KUKA KRL program: EPS_2_25369_MH4A_A_20251128065500.src

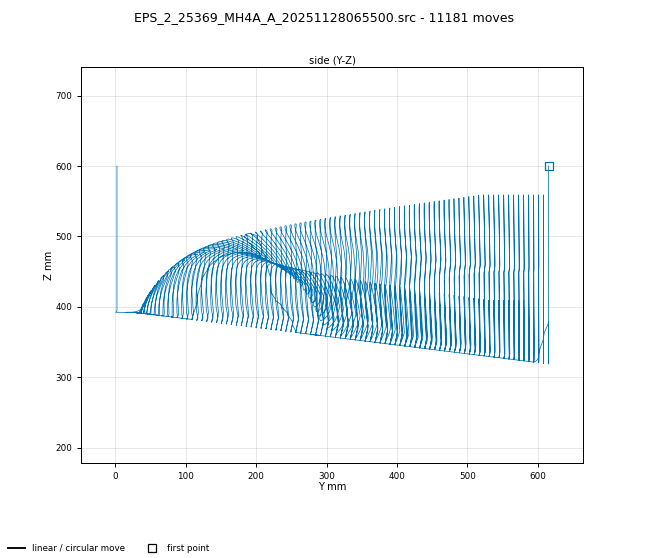
[picture p0: tool path of EPS_2_25369_MH4A_A_20251128065500.src, 11181 of 11183 moves have a stored position in this frame; points joined in program order, loops and branches not executed]
&ACCESS RVP
&REL 4
&COMMENT QRS 19112012
&PARAM EDITMASK = *
DEF PART()
EXT BAS (BAS_COMMAND :IN,REAL :IN )
INT I
BAS (#INITMOV,0 )

;KUKA QRS Post kuka4.cps  Date:22-06-2017 !

File_ID=2934

QRS_PRE_INIT()

;Init var - Until changes are made in qrs_pre_init
Outlet_Square_prg=0
Inlet_1_Square_prg=0
Inlet_2_Square_prg=0
Inlet_3_Square_prg=0
Inlet_4_Square_prg=0
Inlet_5_Square_prg=0

Outlet_1={X 0.000, Y 520.860, Z 458.500, B 0.000, E1 0.000 }
Inlet_1={X 0.000, Y 531.730, Z 308.500, B 0.000, E1 89.000 }
Outlet_1_type=201
Inlet_1_type=201
;QRS#1=Sidecore dimensions
;QRS#2=200-8" PVC SDR 35
;QRS#3=200-8" PVC SDR 35
;QRS#4=
;QRS#5=
;QRS#6=
;QRS#7=
;QRS#8=
;QRS#9=12-08 PSX
;QRS#10=12-08 PSX
;QRS#11=
;QRS#12=
;QRS#13=
;QRS#14=
;QRS#15=
;QRS#16=1220x127x838 2,75'
;QRS#17=EPS Height
;QRS#18=559
;QRS#19=*
;QRS#20= UPDATED VERSION 22-06-2017
;QRS#21=*
Outlet_Square=0100
Inlet_1_Square=0100
Inlet_2_Square=0
Inlet_3_Square=0
Inlet_4_Square=0
Inlet_5_Square=0
Mill_Square=1
Outlet_Square_Prg=204
Inlet_1_Square_prg=204

QRS_INIT()

$ADVANCE=5

; T1
PTP {E1 173.485,E2 173.485}
PTP {X 0,Y 615.499,A -85,B 0,C 180,E1 173.485,E2 173.485,E3 0,E4 0,E5 0,E6 0}
QRS_SPEED_INIT()
LIN {X 0,Y 615.499,Z 600,A -85,B 0,C 180,E1 173.485,E2 173.485,E3 0,E4 0,E5 0,E6 0} C_VEL
LIN {X 0,Y 615.499,Z 392.663,A -85,B 0,C 180,E1 173.485,E2 173.485} C_VEL
LIN {X 0,Y 615.499,Z 380.744,A -85,B 0,C 180,E1 173.485,E2 173.485} C_VEL
LIN {X 0,Y 615.497,Z 379.208,A -85,B 0,C 180,E1 173.418,E2 173.418} C_VEL
LIN {X 0,Y 615.498,Z 369.663,A -85,B 0,C 180,E1 172.455,E2 172.455} C_VEL
LIN {X 0,Y 615.497,Z 359.4,A -85,B 0,C 180,E1 171.629,E2 171.629} C_VEL
LIN {X 0,Y 615.486,Z 347.853,A -85,B 0,C 180,E1 170.884,E2 170.884} C_VEL
LIN {X 0,Y 615.482,Z 336.334,A -85,B 0,C 180,E1 170.304,E2 170.304} C_VEL
LIN {X 0,Y 615.493,Z 324.409,A -85,B 0,C 180,E1 169.847,E2 169.847} C_VEL
LIN {X 0,Y 615.489,Z 318.699,A -85,B 0,C 180,E1 169.66,E2 169.66} C_VEL
LIN {X 0,Y 615.494,Z 318.687,A -85,B 0,C 180,E1 166.799,E2 166.799} C_VEL
LIN {X 0,Y 615.488,Z 318.692,A -85,B 0,C 180,E1 164.095,E2 164.095} C_VEL
LIN {X 0,Y 615.477,Z 318.693,A -85,B 0,C 180,E1 161.354,E2 161.354} C_VEL
LIN {X 0,Y 615.479,Z 318.69,A -85,B 0,C 180,E1 158.568,E2 158.568} C_VEL
LIN {X 0,Y 615.496,Z 318.696,A -85,B 0,C 180,E1 155.728,E2 155.728} C_VEL
LIN {X 0,Y 615.491,Z 318.686,A -85,B 0,C 180,E1 152.823,E2 152.823} C_VEL
LIN {X 0,Y 615.488,Z 318.69,A -85,B 0,C 180,E1 149.84,E2 149.84} C_VEL
LIN {X 0,Y 615.477,Z 318.689,A -85,B 0,C 180,E1 147.542,E2 147.542} C_VEL
LIN {X 0,Y 615.49,Z 318.695,A -85,B 0,C 180,E1 145.185,E2 145.185} C_VEL
LIN {X 0,Y 615.479,Z 318.692,A -85,B 0,C 180,E1 142.757,E2 142.757} C_VEL
LIN {X 0,Y 615.493,Z 318.694,A -85,B 0,C 180,E1 139.911,E2 139.911} C_VEL
LIN {X 0,Y 615.483,Z 318.688,A -85,B 0,C 180,E1 136.954,E2 136.954} C_VEL
LIN {X 0,Y 615.482,Z 318.693,A -85,B 0,C 180,E1 133.997,E2 133.997} C_VEL
LIN {X 0,Y 615.488,Z 318.687,A -85,B 0,C 180,E1 131.474,E2 131.474} C_VEL
LIN {X 0,Y 615.489,Z 318.698,A -85,B 0,C 180,E1 128.905,E2 128.905} C_VEL
LIN {X 0,Y 615.485,Z 318.687,A -85,B 0,C 180,E1 126.425,E2 126.425} C_VEL
LIN {X 0,Y 615.498,Z 318.694,A -85,B 0,C 180,E1 123.536,E2 123.536} C_VEL
LIN {X 0,Y 615.478,Z 318.689,A -85,B 0,C 180,E1 120.92,E2 120.92} C_VEL
LIN {X 0,Y 615.498,Z 318.7,A -85,B 0,C 180,E1 118.452,E2 118.452} C_VEL
LIN {X 0,Y 615.498,Z 318.685,A -85,B 0,C 180,E1 115.571,E2 115.571} C_VEL
LIN {X 0,Y 615.493,Z 318.693,A -85,B 0,C 180,E1 112.844,E2 112.844} C_VEL
LIN {X 0,Y 615.479,Z 318.692,A -85,B 0,C 180,E1 110.033,E2 110.033} C_VEL
LIN {X 0,Y 615.477,Z 318.691,A -85,B 0,C 180,E1 107.271,E2 107.271} C_VEL
LIN {X 0,Y 615.494,Z 318.693,A -85,B 0,C 180,E1 104.549,E2 104.549} C_VEL
LIN {X 0,Y 615.489,Z 318.687,A -85,B 0,C 180,E1 101.861,E2 101.861} C_VEL
LIN {X 0,Y 615.483,Z 318.696,A -85,B 0,C 180,E1 99.199,E2 99.199} C_VEL
LIN {X 0,Y 615.479,Z 318.69,A -85,B 0,C 180,E1 96.557,E2 96.557} C_VEL
LIN {X 0,Y 615.491,Z 318.693,A -85,B 0,C 180,E1 93.928,E2 93.928} C_VEL
LIN {X 0,Y 615.48,Z 318.69,A -85,B 0,C 180,E1 91.309,E2 91.309} C_VEL
LIN {X 0,Y 615.489,Z 318.692,A -85,B 0,C 180,E1 88.691,E2 88.691} C_VEL
LIN {X 0,Y 615.49,Z 318.689,A -85,B 0,C 180,E1 86.071,E2 86.071} C_VEL
LIN {X 0,Y 615.48,Z 318.693,A -85,B 0,C 180,E1 83.428,E2 83.428} C_VEL
LIN {X 0,Y 615.479,Z 318.692,A -85,B 0,C 180,E1 80.801,E2 80.801} C_VEL
LIN {X 0,Y 615.491,Z 318.69,A -85,B 0,C 180,E1 78.139,E2 78.139} C_VEL
LIN {X 0,Y 615.485,Z 318.69,A -85,B 0,C 180,E1 75.451,E2 75.451} C_VEL
LIN {X 0,Y 615.479,Z 318.695,A -85,B 0,C 180,E1 72.729,E2 72.729} C_VEL
LIN {X 0,Y 615.479,Z 318.689,A -85,B 0,C 180,E1 69.967,E2 69.967} C_VEL
LIN {X 0,Y 615.494,Z 318.699,A -85,B 0,C 180,E1 67.155,E2 67.155} C_VEL
LIN {X 0,Y 615.488,Z 318.687,A -85,B 0,C 180,E1 64.284,E2 64.284} C_VEL
LIN {X 0,Y 615.486,Z 318.691,A -85,B 0,C 180,E1 61.342,E2 61.342} C_VEL
LIN {X 0,Y 615.479,Z 318.689,A -85,B 0,C 180,E1 58.915,E2 58.915} C_VEL
LIN {X 0,Y 615.498,Z 318.7,A -85,B 0,C 180,E1 56.464,E2 56.464} C_VEL
LIN {X 0,Y 615.488,Z 318.688,A -85,B 0,C 180,E1 53.575,E2 53.575} C_VEL
LIN {X 0,Y 615.494,Z 318.694,A -85,B 0,C 180,E1 50.937,E2 50.937} C_VEL
LIN {X 0,Y 615.487,Z 318.686,A -85,B 0,C 180,E1 48.526,E2 48.526} C_VEL
LIN {X 0,Y 615.497,Z 318.701,A -85,B 0,C 180,E1 45.851,E2 45.851} C_VEL
LIN {X 0,Y 615.483,Z 318.688,A -85,B 0,C 180,E1 43.046,E2 43.046} C_VEL
LIN {X 0,Y 615.493,Z 318.7,A -85,B 0,C 180,E1 40.606,E2 40.606} C_VEL
LIN {X 0,Y 615.483,Z 318.688,A -85,B 0,C 180,E1 38.011,E2 38.011} C_VEL
LIN {X 0,Y 615.487,Z 318.692,A -85,B 0,C 180,E1 35.616,E2 35.616} C_VEL
LIN {X 0,Y 615.492,Z 318.694,A -85,B 0,C 180,E1 33.236,E2 33.236} C_VEL
LIN {X 0,Y 615.488,Z 318.686,A -85,B 0,C 180,E1 30.92,E2 30.92} C_VEL
LIN {X 0,Y 615.485,Z 318.695,A -85,B 0,C 180,E1 28.449,E2 28.449} C_VEL
LIN {X 0,Y 615.478,Z 318.689,A -85,B 0,C 180,E1 25.716,E2 25.716} C_VEL
LIN {X 0,Y 615.473,Z 318.69,A -85,B 0,C 180,E1 23.557,E2 23.557} C_VEL
LIN {X 0,Y 615.48,Z 318.694,A -85,B 0,C 180,E1 21.432,E2 21.432} C_VEL
LIN {X 0,Y 615.476,Z 318.69,A -85,B 0,C 180,E1 18.646,E2 18.646} C_VEL
LIN {X 0,Y 615.491,Z 318.697,A -85,B 0,C 180,E1 15.905,E2 15.905} C_VEL
LIN {X 0,Y 615.494,Z 318.685,A -85,B 0,C 180,E1 13.201,E2 13.201} C_VEL
LIN {X 0,Y 615.495,Z 318.699,A -85,B 0,C 180,E1 10.527,E2 10.527} C_VEL
LIN {X 0,Y 615.478,Z 318.689,A -85,B 0,C 180,E1 7.876,E2 7.876} C_VEL
LIN {X 0,Y 615.495,Z 318.698,A -85,B 0,C 180,E1 5.241,E2 5.241} C_VEL
LIN {X 0,Y 615.488,Z 318.687,A -85,B 0,C 180,E1 2.618,E2 2.618} C_VEL
LIN {X 0,Y 615.493,Z 318.696,A -85,B 0,C 180,E1 0,E2 0} C_VEL
LIN {X 0,Y 615.488,Z 318.687,A -85,B 0,C 180,E1 -2.618,E2 -2.618} C_VEL
LIN {X 0,Y 615.487,Z 318.696,A -85,B 0,C 180,E1 -5.241,E2 -5.241} C_VEL
LIN {X 0,Y 615.478,Z 318.69,A -85,B 0,C 180,E1 -7.876,E2 -7.876} C_VEL
LIN {X 0,Y 615.495,Z 318.693,A -85,B 0,C 180,E1 -10.527,E2 -10.527} C_VEL
LIN {X 0,Y 615.494,Z 318.686,A -85,B 0,C 180,E1 -13.201,E2 -13.201} C_VEL
LIN {X 0,Y 615.485,Z 318.697,A -85,B 0,C 180,E1 -15.905,E2 -15.905} C_VEL
LIN {X 0,Y 615.477,Z 318.689,A -85,B 0,C 180,E1 -18.647,E2 -18.647} C_VEL
LIN {X 0,Y 615.497,Z 318.7,A -85,B 0,C 180,E1 -21.432,E2 -21.432} C_VEL
LIN {X 0,Y 615.489,Z 318.687,A -85,B 0,C 180,E1 -24.272,E2 -24.272} C_VEL
LIN {X 0,Y 615.489,Z 318.69,A -85,B 0,C 180,E1 -27.177,E2 -27.177} C_VEL
LIN {X 0,Y 615.485,Z 318.691,A -85,B 0,C 180,E1 -29.793,E2 -29.793} C_VEL
LIN {X 0,Y 615.477,Z 318.693,A -85,B 0,C 180,E1 -32.458,E2 -32.458} C_VEL
LIN {X 0,Y 615.491,Z 318.686,A -85,B 0,C 180,E1 -34.815,E2 -34.815} C_VEL
LIN {X 0,Y 615.493,Z 318.699,A -85,B 0,C 180,E1 -37.242,E2 -37.242} C_VEL
LIN {X 0,Y 615.483,Z 318.688,A -85,B 0,C 180,E1 -40.088,E2 -40.088} C_VEL
LIN {X 0,Y 615.486,Z 318.694,A -85,B 0,C 180,E1 -42.353,E2 -42.353} C_VEL
LIN {X 0,Y 615.48,Z 318.689,A -85,B 0,C 180,E1 -45.069,E2 -45.069} C_VEL
LIN {X 0,Y 615.495,Z 318.7,A -85,B 0,C 180,E1 -47.919,E2 -47.919} C_VEL
LIN {X 0,Y 615.477,Z 318.691,A -85,B 0,C 180,E1 -50.249,E2 -50.249} C_VEL
LIN {X 0,Y 615.489,Z 318.696,A -85,B 0,C 180,E1 -53.064,E2 -53.064} C_VEL
LIN {X 0,Y 615.489,Z 318.844,A -85,B 0,C 180,E1 -54.535,E2 -54.535} C_VEL
LIN {X 0,Y 615.495,Z 333.506,A -85,B 0,C 180,E1 -57.349,E2 -57.349} C_VEL
LIN {X 0,Y 615.481,Z 348.225,A -85,B 0,C 180,E1 -60.207,E2 -60.207} C_VEL
LIN {X 0,Y 615.49,Z 362.677,A -85,B 0,C 180,E1 -62.955,E2 -62.955} C_VEL
LIN {X 0,Y 615.48,Z 377.615,A -85,B 0,C 180,E1 -65.727,E2 -65.727} C_VEL
LIN {X 0,Y 615.497,Z 391.289,A -85,B 0,C 180,E1 -68.216,E2 -68.216} C_VEL
LIN {X 0,Y 615.49,Z 406.905,A -85,B 0,C 180,E1 -71.008,E2 -71.008} C_VEL
LIN {X 0,Y 615.485,Z 422.946,A -85,B 0,C 180,E1 -73.831,E2 -73.831} C_VEL
LIN {X 0,Y 615.493,Z 438.092,A -85,B 0,C 180,E1 -76.462,E2 -76.462} C_VEL
LIN {X 0,Y 615.49,Z 448.927,A -85,B 0,C 180,E1 -78.327,E2 -78.327} C_VEL
LIN {X 0,Y 615.479,Z 462.236,A -85,B 0,C 180,E1 -78.556,E2 -78.556} C_VEL
LIN {X 0,Y 615.48,Z 475.326,A -85,B 0,C 180,E1 -78.922,E2 -78.922} C_VEL
LIN {X 0,Y 615.485,Z 487.123,A -85,B 0,C 180,E1 -79.383,E2 -79.383} C_VEL
LIN {X 0,Y 615.486,Z 498.573,A -85,B 0,C 180,E1 -79.972,E2 -79.972} C_VEL
LIN {X 0,Y 615.499,Z 510.019,A -85,B 0,C 180,E1 -80.718,E2 -80.718} C_VEL
LIN {X 0,Y 615.498,Z 519.256,A -85,B 0,C 180,E1 -81.463,E2 -81.463} C_VEL
LIN {X 0,Y 615.499,Z 527.652,A -85,B 0,C 180,E1 -82.29,E2 -82.29} C_VEL
LIN {X 0,Y 615.497,Z 535.69,A -85,B 0,C 180,E1 -83.259,E2 -83.259} C_VEL
LIN {X 0,Y 615.499,Z 541.422,A -85,B 0,C 180,E1 -84.101,E2 -84.101} C_VEL
LIN {X 0,Y 615.496,Z 546.872,A -85,B 0,C 180,E1 -85.087,E2 -85.087} C_VEL
LIN {X 0,Y 615.496,Z 551.141,A -85,B 0,C 180,E1 -86.071,E2 -86.071} C_VEL
LIN {X 0,Y 615.495,Z 553.398,A -85,B 0,C 180,E1 -86.727,E2 -86.727} C_VEL
LIN {X 0,Y 615.497,Z 555.233,A -85,B 0,C 180,E1 -87.382,E2 -87.382} C_VEL
LIN {X 0,Y 615.499,Z 556.607,A -85,B 0,C 180,E1 -88.037,E2 -88.037} C_VEL
LIN {X 0,Y 615.496,Z 558.173,A -85,B 0,C 180,E1 -89.346,E2 -89.346} C_VEL
LIN {X 0,Y 615.494,Z 558.389,A -85,B 0,C 180,E1 -90,E2 -90} C_VEL
LIN {X 0,Y 615.496,Z 557.58,A -85,B 0,C 180,E1 -91.309,E2 -91.309} C_VEL
LIN {X 0,Y 615.499,Z 556.608,A -85,B 0,C 180,E1 -91.963,E2 -91.963} C_VEL
LIN {X 0,Y 615.497,Z 555.233,A -85,B 0,C 180,E1 -92.618,E2 -92.618} C_VEL
LIN {X 0,Y 615.496,Z 552.349,A -85,B 0,C 180,E1 -93.601,E2 -93.601} C_VEL
LIN {X 0,Y 615.498,Z 548.441,A -85,B 0,C 180,E1 -94.584,E2 -94.584} C_VEL
LIN {X 0,Y 615.499,Z 543.405,A -85,B 0,C 180,E1 -95.57,E2 -95.57} C_VEL
LIN {X 0,Y 615.497,Z 536.87,A -85,B 0,C 180,E1 -96.583,E2 -96.583} C_VEL
LIN {X 0,Y 615.497,Z 529.133,A -85,B 0,C 180,E1 -97.545,E2 -97.545} C_VEL
LIN {X 0,Y 615.498,Z 521.045,A -85,B 0,C 180,E1 -98.371,E2 -98.371} C_VEL
LIN {X 0,Y 615.499,Z 511.167,A -85,B 0,C 180,E1 -99.199,E2 -99.199} C_VEL
LIN {X 0,Y 615.491,Z 499.98,A -85,B 0,C 180,E1 -99.945,E2 -99.945} C_VEL
LIN {X 0,Y 615.481,Z 489.022,A -85,B 0,C 180,E1 -100.527,E2 -100.527} C_VEL
LIN {X 0,Y 615.484,Z 476.486,A -85,B 0,C 180,E1 -101.04,E2 -101.04} C_VEL
LIN {X 0,Y 615.478,Z 464.064,A -85,B 0,C 180,E1 -101.402,E2 -101.402} C_VEL
LIN {X 0,Y 615.488,Z 450.461,A -85,B 0,C 180,E1 -101.652,E2 -101.652} C_VEL
LIN {X 0,Y 615.49,Z 448.798,A -85,B 0,C 180,E1 -101.694,E2 -101.694} C_VEL
LIN {X 0,Y 615.483,Z 432.25,A -85,B 0,C 180,E1 -104.549,E2 -104.549} C_VEL
LIN {X 0,Y 615.478,Z 416.659,A -85,B 0,C 180,E1 -107.271,E2 -107.271} C_VEL
LIN {X 0,Y 615.479,Z 401.052,A -85,B 0,C 180,E1 -110.033,E2 -110.033} C_VEL
LIN {X 0,Y 615.492,Z 385.431,A -85,B 0,C 180,E1 -112.845,E2 -112.845} C_VEL
LIN {X 0,Y 615.492,Z 369.796,A -85,B 0,C 180,E1 -115.716,E2 -115.716} C_VEL
LIN {X 0,Y 615.491,Z 355.237,A -85,B 0,C 180,E1 -118.45,E2 -118.45} C_VEL
LIN {X 0,Y 615.485,Z 341.563,A -85,B 0,C 180,E1 -121.085,E2 -121.085} C_VEL
LIN {X 0,Y 615.49,Z 333.379,A -85,B 0,C 180,E1 -122.652,E2 -122.652} C_VEL
LIN {X 0,Y 615.481,Z 318.694,A -85,B 0,C 180,E1 -125.215,E2 -125.215} C_VEL
LIN {X 0,Y 615.483,Z 318.694,A -85,B 0,C 180,E1 -128.069,E2 -128.069} C_VEL
LIN {X 0,Y 615.482,Z 318.696,A -85,B 0,C 180,E1 -130.607,E2 -130.607} C_VEL
LIN {X 0,Y 615.498,Z 318.696,A -85,B 0,C 180,E1 -133.244,E2 -133.244} C_VEL
LIN {X 0,Y 615.494,Z 318.698,A -85,B 0,C 180,E1 -136.002,E2 -136.002} C_VEL
LIN {X 0,Y 615.494,Z 318.696,A -85,B 0,C 180,E1 -138.905,E2 -138.905} C_VEL
LIN {X 0,Y 615.492,Z 318.693,A -85,B 0,C 180,E1 -141.096,E2 -141.096} C_VEL
LIN {X 0,Y 615.478,Z 318.695,A -85,B 0,C 180,E1 -143.574,E2 -143.574} C_VEL
LIN {X 0,Y 615.494,Z 318.695,A -85,B 0,C 180,E1 -145.978,E2 -145.978} C_VEL
LIN {X 0,Y 615.489,Z 318.694,A -85,B 0,C 180,E1 -148.915,E2 -148.915} C_VEL
LIN {X 0,Y 615.491,Z 318.697,A -85,B 0,C 180,E1 -151.55,E2 -151.55} C_VEL
LIN {X 0,Y 615.485,Z 318.7,A -85,B 0,C 180,E1 -154.284,E2 -154.284} C_VEL
LIN {X 0,Y 615.474,Z 318.696,A -85,B 0,C 180,E1 -156.443,E2 -156.443} C_VEL
LIN {X 0,Y 615.495,Z 318.696,A -85,B 0,C 180,E1 -158.568,E2 -158.568} C_VEL
LIN {X 0,Y 615.489,Z 318.697,A -85,B 0,C 180,E1 -161.396,E2 -161.396} C_VEL
LIN {X 0,Y 615.488,Z 318.7,A -85,B 0,C 180,E1 -164.095,E2 -164.095} C_VEL
LIN {X 0,Y 615.498,Z 318.7,A -85,B 0,C 180,E1 -166.799,E2 -166.799} C_VEL
LIN {X 0,Y 615.497,Z 318.692,A -85,B 0,C 180,E1 -167.763,E2 -167.763} C_VEL
LIN {X 0,Y 615.493,Z 331.231,A -85,B 0,C 180,E1 -168.181,E2 -168.181} C_VEL
LIN {X 0,Y 615.492,Z 343.212,A -85,B 0,C 180,E1 -168.723,E2 -168.723} C_VEL
LIN {X 0,Y 615.483,Z 354.543,A -85,B 0,C 180,E1 -169.384,E2 -169.384} C_VEL
LIN {X 0,Y 615.499,Z 364.889,A -85,B 0,C 180,E1 -170.138,E2 -170.138} C_VEL
LIN {X 0,Y 615.497,Z 374.108,A -85,B 0,C 180,E1 -170.967,E2 -170.967} C_VEL
LIN {X 0,Y 615.498,Z 383.029,A -85,B 0,C 180,E1 -171.959,E2 -171.959} C_VEL
LIN {X 0,Y 615.497,Z 390.162,A -85,B 0,C 180,E1 -172.943,E2 -172.943} C_VEL
LIN {X 0,Y 615.498,Z 395.032,A -85,B 0,C 180,E1 -173.772,E2 -173.772} C_VEL
LIN {X 0,Y 615.495,Z 399.723,A -85,B 0,C 180,E1 -174.759,E2 -174.759} C_VEL
LIN {X 0,Y 615.496,Z 403.307,A -85,B 0,C 180,E1 -175.743,E2 -175.743} C_VEL
LIN {X 0,Y 615.496,Z 405.895,A -85,B 0,C 180,E1 -176.727,E2 -176.727} C_VEL
LIN {X 0,Y 615.497,Z 407.108,A -85,B 0,C 180,E1 -177.382,E2 -177.382} C_VEL
LIN {X 0,Y 615.496,Z 407.923,A -85,B 0,C 180,E1 -178.037,E2 -178.037} C_VEL
LIN {X 0,Y 615.495,Z 408.323,A -85,B 0,C 180,E1 -179.346,E2 -179.346} C_VEL
LIN {X 0,Y 615.495,Z 407.962,A -85,B 0,C 180,E1 -180,E2 -180} C_VEL
LIN {X 0,Y 615.496,Z 407.198,A -85,B 0,C 180,E1 -180.654,E2 -180.654} C_VEL
LIN {X 0,Y 615.499,Z 404.43,A -85,B 0,C 180,E1 -181.963,E2 -181.963} C_VEL
LIN {X 0,Y 615.496,Z 401.246,A -85,B 0,C 180,E1 -182.945,E2 -182.945} C_VEL
LIN {X 0,Y 615.495,Z 397.016,A -85,B 0,C 180,E1 -183.928,E2 -183.928} C_VEL
LIN {X 0,Y 615.497,Z 390.61,A -85,B 0,C 180,E1 -185.077,E2 -185.077} C_VEL
LIN {X 0,Y 615.497,Z 383.586,A -85,B 0,C 180,E1 -186.063,E2 -186.063} C_VEL
LIN {X 0,Y 615.497,Z 379.208,A -85,B 0,C 180,E1 -186.582,E2 -186.582} C_VEL
LIN {X 0,Y 614.836,Z 375.55,A -85,B 0,C 180,E1 -186.998,E2 -186.998} C_VEL
LIN {X 0,Y 612.016,Z 369.242,A -85,B 0,C 180,E1 -187.656,E2 -187.656} C_VEL
LIN {X 0,Y 609.167,Z 362.269,A -85,B 0,C 180,E1 -188.273,E2 -188.273} C_VEL
LIN {X 0,Y 608.486,Z 357.621,A -85,B 0,C 180,E1 -188.624,E2 -188.624} C_VEL
LIN {X 0,Y 608.506,Z 346.75,A -85,B 0,C 180,E1 -189.305,E2 -189.305} C_VEL
LIN {X 0,Y 608.516,Z 334.78,A -85,B 0,C 180,E1 -189.892,E2 -189.892} C_VEL
LIN {X 0,Y 608.541,Z 322.302,A -85,B 0,C 180,E1 -190.354,E2 -190.354} C_VEL
LIN {X 0,Y 608.462,Z 319.694,A -85,B 0,C 180,E1 -190.439,E2 -190.439} C_VEL
LIN {X 0,Y 608.472,Z 319.69,A -85,B 0,C 180,E1 -193.356,E2 -193.356} C_VEL
LIN {X 0,Y 608.462,Z 319.69,A -85,B 0,C 180,E1 -196.094,E2 -196.094} C_VEL
LIN {X 0,Y 608.455,Z 319.694,A -85,B 0,C 180,E1 -198.87,E2 -198.87} C_VEL
LIN {X 0,Y 608.469,Z 319.688,A -85,B 0,C 180,E1 -201.691,E2 -201.691} C_VEL
LIN {X 0,Y 608.462,Z 319.694,A -85,B 0,C 180,E1 -204.571,E2 -204.571} C_VEL
LIN {X 0,Y 608.454,Z 319.692,A -85,B 0,C 180,E1 -207.518,E2 -207.518} C_VEL
LIN {X 0,Y 608.475,Z 319.691,A -85,B 0,C 180,E1 -209.972,E2 -209.972} C_VEL
LIN {X 0,Y 608.455,Z 319.689,A -85,B 0,C 180,E1 -212.521,E2 -212.521} C_VEL
LIN {X 0,Y 608.454,Z 319.696,A -85,B 0,C 180,E1 -214.905,E2 -214.905} C_VEL
LIN {X 0,Y 608.469,Z 319.687,A -85,B 0,C 180,E1 -217.746,E2 -217.746} C_VEL
LIN {X 0,Y 608.458,Z 319.698,A -85,B 0,C 180,E1 -220.329,E2 -220.329} C_VEL
LIN {X 0,Y 608.45,Z 319.69,A -85,B 0,C 180,E1 -222.96,E2 -222.96} C_VEL
LIN {X 0,Y 608.46,Z 319.696,A -85,B 0,C 180,E1 -225.736,E2 -225.736} C_VEL
LIN {X 0,Y 608.466,Z 319.689,A -85,B 0,C 180,E1 -228.657,E2 -228.657} C_VEL
LIN {X 0,Y 608.465,Z 319.688,A -85,B 0,C 180,E1 -231.76,E2 -231.76} C_VEL
LIN {X 0,Y 608.448,Z 319.691,A -85,B 0,C 180,E1 -233.954,E2 -233.954} C_VEL
LIN {X 0,Y 608.472,Z 319.695,A -85,B 0,C 180,E1 -236.33,E2 -236.33} C_VEL
LIN {X 0,Y 608.448,Z 319.69,A -85,B 0,C 180,E1 -238.732,E2 -238.732} C_VEL
LIN {X 0,Y 608.478,Z 319.692,A -85,B 0,C 180,E1 -241.379,E2 -241.379} C_VEL
LIN {X 0,Y 608.476,Z 319.687,A -85,B 0,C 180,E1 -244.278,E2 -244.278} C_VEL
LIN {X 0,Y 608.456,Z 319.698,A -85,B 0,C 180,E1 -246.876,E2 -246.876} C_VEL
LIN {X 0,Y 608.468,Z 319.688,A -85,B 0,C 180,E1 -249.321,E2 -249.321} C_VEL
LIN {X 0,Y 608.447,Z 319.693,A -85,B 0,C 180,E1 -251.828,E2 -251.828} C_VEL
LIN {X 0,Y 608.468,Z 319.688,A -85,B 0,C 180,E1 -254.594,E2 -254.594} C_VEL
LIN {X 0,Y 608.479,Z 319.692,A -85,B 0,C 180,E1 -257.323,E2 -257.323} C_VEL
LIN {X 0,Y 608.465,Z 319.688,A -85,B 0,C 180,E1 -260.023,E2 -260.023} C_VEL
LIN {X 0,Y 608.469,Z 319.694,A -85,B 0,C 180,E1 -262.701,E2 -262.701} C_VEL
LIN {X 0,Y 608.45,Z 319.69,A -85,B 0,C 180,E1 -265.362,E2 -265.362} C_VEL
LIN {X 0,Y 608.469,Z 319.694,A -85,B 0,C 180,E1 -268.014,E2 -268.014} C_VEL
LIN {X 0,Y 608.475,Z 319.687,A -85,B 0,C 180,E1 -270.662,E2 -270.662} C_VEL
LIN {X 0,Y 608.487,Z 319.692,A -85,B 0,C 180,E1 -273.311,E2 -273.311} C_VEL
LIN {X 0,Y 608.492,Z 319.685,A -85,B 0,C 180,E1 -275.967,E2 -275.967} C_VEL
LIN {X 0,Y 608.457,Z 319.696,A -85,B 0,C 180,E1 -278.636,E2 -278.636} C_VEL
LIN {X 0,Y 608.456,Z 319.689,A -85,B 0,C 180,E1 -281.324,E2 -281.324} C_VEL
LIN {X 0,Y 608.472,Z 319.696,A -85,B 0,C 180,E1 -284.038,E2 -284.038} C_VEL
LIN {X 0,Y 608.476,Z 319.687,A -85,B 0,C 180,E1 -286.784,E2 -286.784} C_VEL
LIN {X 0,Y 608.454,Z 319.695,A -85,B 0,C 180,E1 -289.571,E2 -289.571} C_VEL
LIN {X 0,Y 608.479,Z 319.688,A -85,B 0,C 180,E1 -292.405,E2 -292.405} C_VEL
LIN {X 0,Y 608.455,Z 319.69,A -85,B 0,C 180,E1 -295.301,E2 -295.301} C_VEL
LIN {X 0,Y 608.447,Z 319.691,A -85,B 0,C 180,E1 -297.518,E2 -297.518} C_VEL
LIN {X 0,Y 608.475,Z 319.696,A -85,B 0,C 180,E1 -299.973,E2 -299.973} C_VEL
LIN {X 0,Y 608.459,Z 319.689,A -85,B 0,C 180,E1 -302.88,E2 -302.88} C_VEL
LIN {X 0,Y 608.44,Z 319.7,A -85,B 0,C 180,E1 -305.278,E2 -305.278} C_VEL
LIN {X 0,Y 608.468,Z 319.688,A -85,B 0,C 180,E1 -307.747,E2 -307.747} C_VEL
LIN {X 0,Y 608.452,Z 319.694,A -85,B 0,C 180,E1 -310.329,E2 -310.329} C_VEL
LIN {X 0,Y 608.483,Z 319.686,A -85,B 0,C 180,E1 -313.31,E2 -313.31} C_VEL
LIN {X 0,Y 608.479,Z 319.691,A -85,B 0,C 180,E1 -316.131,E2 -316.131} C_VEL
LIN {X 0,Y 608.451,Z 319.69,A -85,B 0,C 180,E1 -318.823,E2 -318.823} C_VEL
LIN {X 0,Y 608.466,Z 319.689,A -85,B 0,C 180,E1 -321.761,E2 -321.761} C_VEL
LIN {X 0,Y 608.452,Z 319.69,A -85,B 0,C 180,E1 -323.955,E2 -323.955} C_VEL
LIN {X 0,Y 608.472,Z 319.692,A -85,B 0,C 180,E1 -326.33,E2 -326.33} C_VEL
LIN {X 0,Y 608.451,Z 319.692,A -85,B 0,C 180,E1 -328.733,E2 -328.733} C_VEL
LIN {X 0,Y 608.473,Z 319.689,A -85,B 0,C 180,E1 -331.381,E2 -331.381} C_VEL
LIN {X 0,Y 608.446,Z 319.694,A -85,B 0,C 180,E1 -333.965,E2 -333.965} C_VEL
LIN {X 0,Y 608.465,Z 319.688,A -85,B 0,C 180,E1 -336.155,E2 -336.155} C_VEL
LIN {X 0,Y 608.452,Z 319.697,A -85,B 0,C 180,E1 -339.018,E2 -339.018} C_VEL
LIN {X 0,Y 608.447,Z 319.691,A -85,B 0,C 180,E1 -341.828,E2 -341.828} C_VEL
LIN {X 0,Y 608.476,Z 319.69,A -85,B 0,C 180,E1 -344.594,E2 -344.594} C_VEL
LIN {X 0,Y 608.476,Z 319.689,A -85,B 0,C 180,E1 -347.323,E2 -347.323} C_VEL
LIN {X 0,Y 608.452,Z 319.691,A -85,B 0,C 180,E1 -350.023,E2 -350.023} C_VEL
LIN {X 0,Y 608.47,Z 319.69,A -85,B 0,C 180,E1 -352.701,E2 -352.701} C_VEL
LIN {X 0,Y 608.455,Z 319.691,A -85,B 0,C 180,E1 -355.362,E2 -355.362} C_VEL
LIN {X 0,Y 608.451,Z 319.693,A -85,B 0,C 180,E1 -358.014,E2 -358.014} C_VEL
LIN {X 0,Y 608.479,Z 319.688,A -85,B 0,C 180,E1 -360.662,E2 -360.662} C_VEL
LIN {X 0,Y 608.479,Z 319.689,A -85,B 0,C 180,E1 -363.311,E2 -363.311} C_VEL
LIN {X 0,Y 608.456,Z 319.691,A -85,B 0,C 180,E1 -365.967,E2 -365.967} C_VEL
LIN {X 0,Y 608.46,Z 319.692,A -85,B 0,C 180,E1 -368.636,E2 -368.636} C_VEL
LIN {X 0,Y 608.481,Z 319.687,A -85,B 0,C 180,E1 -371.324,E2 -371.324} C_VEL
LIN {X 0,Y 608.453,Z 319.694,A -85,B 0,C 180,E1 -374.038,E2 -374.038} C_VEL
LIN {X 0,Y 608.446,Z 319.691,A -85,B 0,C 180,E1 -376.784,E2 -376.784} C_VEL
LIN {X 0,Y 608.461,Z 319.696,A -85,B 0,C 180,E1 -379.57,E2 -379.57} C_VEL
LIN {X 0,Y 608.465,Z 319.688,A -85,B 0,C 180,E1 -382.476,E2 -382.476} C_VEL
LIN {X 0,Y 608.46,Z 319.692,A -85,B 0,C 180,E1 -384.571,E2 -384.571} C_VEL
LIN {X 0,Y 608.485,Z 319.687,A -85,B 0,C 180,E1 -387.207,E2 -387.207} C_VEL
LIN {X 0,Y 608.471,Z 319.691,A -85,B 0,C 180,E1 -389.971,E2 -389.971} C_VEL
LIN {X 0,Y 608.454,Z 319.689,A -85,B 0,C 180,E1 -392.88,E2 -392.88} C_VEL
LIN {X 0,Y 608.451,Z 319.694,A -85,B 0,C 180,E1 -395.277,E2 -395.277} C_VEL
LIN {X 0,Y 608.471,Z 319.69,A -85,B 0,C 180,E1 -397.746,E2 -397.746} C_VEL
LIN {X 0,Y 608.448,Z 319.691,A -85,B 0,C 180,E1 -400.328,E2 -400.328} C_VEL
LIN {X 0,Y 608.45,Z 319.693,A -85,B 0,C 180,E1 -402.96,E2 -402.96} C_VEL
LIN {X 0,Y 608.464,Z 319.69,A -85,B 0,C 180,E1 -405.736,E2 -405.736} C_VEL
LIN {X 0,Y 608.463,Z 319.689,A -85,B 0,C 180,E1 -408.658,E2 -408.658} C_VEL
LIN {X 0,Y 608.464,Z 319.693,A -85,B 0,C 180,E1 -411.76,E2 -411.76} C_VEL
LIN {X 0,Y 608.475,Z 319.736,A -85,B 0,C 180,E1 -414.318,E2 -414.318} C_VEL
LIN {X 0,Y 608.584,Z 327.953,A -85,B 0,C 180,E1 -415.938,E2 -415.938} C_VEL
LIN {X 0,Y 608.614,Z 342.471,A -85,B 0,C 180,E1 -418.707,E2 -418.707} C_VEL
LIN {X 0,Y 608.593,Z 356.081,A -85,B 0,C 180,E1 -421.36,E2 -421.36} C_VEL
LIN {X 0,Y 608.569,Z 371.344,A -85,B 0,C 180,E1 -424.261,E2 -424.261} C_VEL
LIN {X 0,Y 608.55,Z 387.408,A -85,B 0,C 180,E1 -427.239,E2 -427.239} C_VEL
LIN {X 0,Y 608.509,Z 403.057,A -85,B 0,C 180,E1 -430.08,E2 -430.08} C_VEL
LIN {X 0,Y 608.47,Z 418.709,A -85,B 0,C 180,E1 -432.87,E2 -432.87} C_VEL
LIN {X 0,Y 608.46,Z 434.36,A -85,B 0,C 180,E1 -435.621,E2 -435.621} C_VEL
LIN {X 0,Y 608.448,Z 449.156,A -85,B 0,C 180,E1 -438.19,E2 -438.19} C_VEL
LIN {X 0,Y 608.541,Z 463.261,A -85,B 0,C 180,E1 -438.445,E2 -438.445} C_VEL
LIN {X 0,Y 608.523,Z 475.897,A -85,B 0,C 180,E1 -438.808,E2 -438.808} C_VEL
LIN {X 0,Y 608.515,Z 487.598,A -85,B 0,C 180,E1 -439.275,E2 -439.275} C_VEL
LIN {X 0,Y 608.491,Z 498.753,A -85,B 0,C 180,E1 -439.855,E2 -439.855} C_VEL
LIN {X 0,Y 608.504,Z 510.25,A -85,B 0,C 180,E1 -440.611,E2 -440.611} C_VEL
LIN {X 0,Y 608.472,Z 519.535,A -85,B 0,C 180,E1 -441.364,E2 -441.364} C_VEL
LIN {X 0,Y 608.456,Z 527.988,A -85,B 0,C 180,E1 -442.2,E2 -442.2} C_VEL
LIN {X 0,Y 608.462,Z 536.234,A -85,B 0,C 180,E1 -443.201,E2 -443.201} C_VEL
LIN {X 0,Y 608.437,Z 542.876,A -85,B 0,C 180,E1 -444.199,E2 -444.199} C_VEL
LIN {X 0,Y 608.432,Z 548.95,A -85,B 0,C 180,E1 -445.362,E2 -445.362} C_VEL
LIN {X 0,Y 608.449,Z 552.896,A -85,B 0,C 180,E1 -446.358,E2 -446.358} C_VEL
LIN {X 0,Y 608.425,Z 555.809,A -85,B 0,C 180,E1 -447.352,E2 -447.352} C_VEL
LIN {X 0,Y 608.444,Z 557.201,A -85,B 0,C 180,E1 -448.014,E2 -448.014} C_VEL
LIN {X 0,Y 608.438,Z 558.783,A -85,B 0,C 180,E1 -449.338,E2 -449.338} C_VEL
LIN {X 0,Y 608.434,Z 559,A -85,B 0,C 180,E1 -450,E2 -450} C_VEL
LIN {X 0,Y 608.448,Z 558.184,A -85,B 0,C 180,E1 -451.324,E2 -451.324} C_VEL
LIN {X 0,Y 608.444,Z 557.201,A -85,B 0,C 180,E1 -451.986,E2 -451.986} C_VEL
LIN {X 0,Y 608.425,Z 555.809,A -85,B 0,C 180,E1 -452.648,E2 -452.648} C_VEL
LIN {X 0,Y 608.449,Z 552.896,A -85,B 0,C 180,E1 -453.642,E2 -453.642} C_VEL
LIN {X 0,Y 608.432,Z 548.95,A -85,B 0,C 180,E1 -454.638,E2 -454.638} C_VEL
LIN {X 0,Y 608.437,Z 542.877,A -85,B 0,C 180,E1 -455.801,E2 -455.801} C_VEL
LIN {X 0,Y 608.462,Z 536.235,A -85,B 0,C 180,E1 -456.799,E2 -456.799} C_VEL
LIN {X 0,Y 608.456,Z 527.989,A -85,B 0,C 180,E1 -457.8,E2 -457.8} C_VEL
LIN {X 0,Y 608.472,Z 519.536,A -85,B 0,C 180,E1 -458.636,E2 -458.636} C_VEL
LIN {X 0,Y 608.481,Z 509.09,A -85,B 0,C 180,E1 -459.473,E2 -459.473} C_VEL
LIN {X 0,Y 608.491,Z 498.755,A -85,B 0,C 180,E1 -460.145,E2 -460.145} C_VEL
LIN {X 0,Y 608.517,Z 487.265,A -85,B 0,C 180,E1 -460.74,E2 -460.74} C_VEL
LIN {X 0,Y 608.529,Z 474.892,A -85,B 0,C 180,E1 -461.225,E2 -461.225} C_VEL
LIN {X 0,Y 608.542,Z 461.436,A -85,B 0,C 180,E1 -461.597,E2 -461.597} C_VEL
LIN {X 0,Y 608.448,Z 449.156,A -85,B 0,C 180,E1 -461.81,E2 -461.81} C_VEL
LIN {X 0,Y 608.46,Z 434.361,A -85,B 0,C 180,E1 -464.379,E2 -464.379} C_VEL
LIN {X 0,Y 608.471,Z 418.709,A -85,B 0,C 180,E1 -467.13,E2 -467.13} C_VEL
LIN {X 0,Y 608.509,Z 403.058,A -85,B 0,C 180,E1 -469.92,E2 -469.92} C_VEL
LIN {X 0,Y 608.55,Z 387.408,A -85,B 0,C 180,E1 -472.76,E2 -472.76} C_VEL
LIN {X 0,Y 608.569,Z 371.344,A -85,B 0,C 180,E1 -475.739,E2 -475.739} C_VEL
LIN {X 0,Y 608.593,Z 356.081,A -85,B 0,C 180,E1 -478.64,E2 -478.64} C_VEL
LIN {X 0,Y 608.614,Z 342.391,A -85,B 0,C 180,E1 -481.308,E2 -481.308} C_VEL
LIN {X 0,Y 608.517,Z 324.264,A -85,B 0,C 180,E1 -484.466,E2 -484.466} C_VEL
LIN {X 0,Y 608.472,Z 319.691,A -85,B 0,C 180,E1 -485.301,E2 -485.301} C_VEL
LIN {X 0,Y 608.467,Z 319.691,A -85,B 0,C 180,E1 -488.24,E2 -488.24} C_VEL
LIN {X 0,Y 608.466,Z 319.693,A -85,B 0,C 180,E1 -491.342,E2 -491.342} C_VEL
LIN {X 0,Y 608.459,Z 319.695,A -85,B 0,C 180,E1 -494.264,E2 -494.264} C_VEL
LIN {X 0,Y 608.449,Z 319.696,A -85,B 0,C 180,E1 -497.04,E2 -497.04} C_VEL
LIN {X 0,Y 608.457,Z 319.693,A -85,B 0,C 180,E1 -499.697,E2 -499.697} C_VEL
LIN {X 0,Y 608.473,Z 319.69,A -85,B 0,C 180,E1 -502.254,E2 -502.254} C_VEL
LIN {X 0,Y 608.485,Z 319.689,A -85,B 0,C 180,E1 -505.09,E2 -505.09} C_VEL
LIN {X 0,Y 608.465,Z 319.691,A -85,B 0,C 180,E1 -507.905,E2 -507.905} C_VEL
LIN {X 0,Y 608.47,Z 319.693,A -85,B 0,C 180,E1 -510.22,E2 -510.22} C_VEL
LIN {X 0,Y 608.488,Z 319.693,A -85,B 0,C 180,E1 -512.792,E2 -512.792} C_VEL
LIN {X 0,Y 608.485,Z 319.691,A -85,B 0,C 180,E1 -515.847,E2 -515.847} C_VEL
LIN {X 0,Y 608.477,Z 319.695,A -85,B 0,C 180,E1 -518.309,E2 -518.309} C_VEL
LIN {X 0,Y 608.475,Z 319.694,A -85,B 0,C 180,E1 -521.284,E2 -521.284} C_VEL
LIN {X 0,Y 608.463,Z 319.696,A -85,B 0,C 180,E1 -523.906,E2 -523.906} C_VEL
LIN {X 0,Y 608.47,Z 319.694,A -85,B 0,C 180,E1 -526.644,E2 -526.644} C_VEL
LIN {X 0,Y 608.524,Z 319.886,A -85,B 0,C 180,E1 -527.663,E2 -527.663} C_VEL
LIN {X 0,Y 608.517,Z 332.15,A -85,B 0,C 180,E1 -528.086,E2 -528.086} C_VEL
LIN {X 0,Y 608.492,Z 344.735,A -85,B 0,C 180,E1 -528.676,E2 -528.676} C_VEL
LIN {X 0,Y 608.486,Z 355.936,A -85,B 0,C 180,E1 -529.35,E2 -529.35} C_VEL
LIN {X 0,Y 608.498,Z 366.034,A -85,B 0,C 180,E1 -530.107,E2 -530.107} C_VEL
LIN {X 0,Y 608.473,Z 375.94,A -85,B 0,C 180,E1 -531.029,E2 -531.029} C_VEL
LIN {X 0,Y 608.459,Z 384.652,A -85,B 0,C 180,E1 -532.033,E2 -532.033} C_VEL
LIN {X 0,Y 608.444,Z 391.598,A -85,B 0,C 180,E1 -533.034,E2 -533.034} C_VEL
LIN {X 0,Y 608.437,Z 397.16,A -85,B 0,C 180,E1 -534.033,E2 -534.033} C_VEL
LIN {X 0,Y 608.436,Z 401.524,A -85,B 0,C 180,E1 -535.03,E2 -535.03} C_VEL
LIN {X 0,Y 608.433,Z 404.82,A -85,B 0,C 180,E1 -536.026,E2 -536.026} C_VEL
LIN {X 0,Y 608.424,Z 406.456,A -85,B 0,C 180,E1 -536.689,E2 -536.689} C_VEL
LIN {X 0,Y 608.441,Z 408.52,A -85,B 0,C 180,E1 -538.014,E2 -538.014} C_VEL
LIN {X 0,Y 608.438,Z 408.937,A -85,B 0,C 180,E1 -539.338,E2 -539.338} C_VEL
LIN {X 0,Y 608.435,Z 408.577,A -85,B 0,C 180,E1 -540,E2 -540} C_VEL
LIN {X 0,Y 608.439,Z 407.814,A -85,B 0,C 180,E1 -540.662,E2 -540.662} C_VEL
LIN {X 0,Y 608.449,Z 406.623,A -85,B 0,C 180,E1 -541.324,E2 -541.324} C_VEL
LIN {X 0,Y 608.45,Z 404.081,A -85,B 0,C 180,E1 -542.317,E2 -542.317} C_VEL
LIN {X 0,Y 608.431,Z 400.543,A -85,B 0,C 180,E1 -543.311,E2 -543.311} C_VEL
LIN {X 0,Y 608.441,Z 395.906,A -85,B 0,C 180,E1 -544.306,E2 -544.306} C_VEL
LIN {X 0,Y 608.462,Z 388.91,A -85,B 0,C 180,E1 -545.468,E2 -545.468} C_VEL
LIN {X 0,Y 608.469,Z 381.039,A -85,B 0,C 180,E1 -546.502,E2 -546.502} C_VEL
LIN {X 0,Y 608.472,Z 371.84,A -85,B 0,C 180,E1 -547.466,E2 -547.466} C_VEL
LIN {X 0,Y 608.496,Z 362.041,A -85,B 0,C 180,E1 -548.301,E2 -548.301} C_VEL
LIN {X 0,Y 608.486,Z 357.621,A -85,B 0,C 180,E1 -548.624,E2 -548.624} C_VEL
LIN {X 0,Y 607.798,Z 352.923,A -85,B 0,C 180,E1 -548.958,E2 -548.958} C_VEL
LIN {X 0,Y 604.953,Z 345.102,A -85,B 0,C 180,E1 -549.471,E2 -549.471} C_VEL
LIN {X 0,Y 602.157,Z 336.875,A -85,B 0,C 180,E1 -549.922,E2 -549.922} C_VEL
LIN {X 0,Y 601.541,Z 331.55,A -85,B 0,C 180,E1 -550.157,E2 -550.157} C_VEL
LIN {X 0,Y 601.443,Z 320.567,A -85,B 0,C 180,E1 -550.563,E2 -550.563} C_VEL
LIN {X 0,Y 601.426,Z 320.569,A -85,B 0,C 180,E1 -553.516,E2 -553.516} C_VEL
LIN {X 0,Y 601.441,Z 320.563,A -85,B 0,C 180,E1 -556.287,E2 -556.287} C_VEL
LIN {X 0,Y 601.42,Z 320.574,A -85,B 0,C 180,E1 -559.099,E2 -559.099} C_VEL
LIN {X 0,Y 601.408,Z 320.57,A -85,B 0,C 180,E1 -561.239,E2 -561.239} C_VEL
LIN {X 0,Y 601.464,Z 320.565,A -85,B 0,C 180,E1 -564.14,E2 -564.14} C_VEL
LIN {X 0,Y 601.458,Z 320.561,A -85,B 0,C 180,E1 -567.111,E2 -567.111} C_VEL
LIN {X 0,Y 601.433,Z 320.566,A -85,B 0,C 180,E1 -570.148,E2 -570.148} C_VEL
LIN {X 0,Y 601.42,Z 320.567,A -85,B 0,C 180,E1 -572.714,E2 -572.714} C_VEL
LIN {X 0,Y 601.4,Z 320.575,A -85,B 0,C 180,E1 -575.112,E2 -575.112} C_VEL
LIN {X 0,Y 601.437,Z 320.564,A -85,B 0,C 180,E1 -577.419,E2 -577.419} C_VEL
LIN {X 0,Y 601.416,Z 320.57,A -85,B 0,C 180,E1 -579.995,E2 -579.995} C_VEL
LIN {X 0,Y 601.413,Z 320.568,A -85,B 0,C 180,E1 -582.67,E2 -582.67} C_VEL
LIN {X 0,Y 601.429,Z 320.571,A -85,B 0,C 180,E1 -585.482,E2 -585.482} C_VEL
LIN {X 0,Y 601.428,Z 320.565,A -85,B 0,C 180,E1 -588.406,E2 -588.406} C_VEL
LIN {X 0,Y 601.434,Z 320.565,A -85,B 0,C 180,E1 -591.529,E2 -591.529} C_VEL
LIN {X 0,Y 601.389,Z 320.574,A -85,B 0,C 180,E1 -594.245,E2 -594.245} C_VEL
LIN {X 0,Y 601.432,Z 320.566,A -85,B 0,C 180,E1 -596.687,E2 -596.687} C_VEL
LIN {X 0,Y 601.416,Z 320.566,A -85,B 0,C 180,E1 -599.058,E2 -599.058} C_VEL
LIN {X 0,Y 601.437,Z 320.569,A -85,B 0,C 180,E1 -601.373,E2 -601.373} C_VEL
LIN {X 0,Y 601.415,Z 320.566,A -85,B 0,C 180,E1 -604.132,E2 -604.132} C_VEL
LIN {X 0,Y 601.422,Z 320.569,A -85,B 0,C 180,E1 -606.59,E2 -606.59} C_VEL
LIN {X 0,Y 601.431,Z 320.564,A -85,B 0,C 180,E1 -609.478,E2 -609.478} C_VEL
LIN {X 0,Y 601.393,Z 320.576,A -85,B 0,C 180,E1 -612.311,E2 -612.311} C_VEL
LIN {X 0,Y 601.415,Z 320.568,A -85,B 0,C 180,E1 -614.409,E2 -614.409} C_VEL
LIN {X 0,Y 601.423,Z 320.569,A -85,B 0,C 180,E1 -617.172,E2 -617.172} C_VEL
LIN {X 0,Y 601.441,Z 320.564,A -85,B 0,C 180,E1 -619.905,E2 -619.905} C_VEL
LIN {X 0,Y 601.445,Z 320.568,A -85,B 0,C 180,E1 -622.615,E2 -622.615} C_VEL
LIN {X 0,Y 601.42,Z 320.566,A -85,B 0,C 180,E1 -625.308,E2 -625.308} C_VEL
LIN {X 0,Y 601.437,Z 320.57,A -85,B 0,C 180,E1 -627.991,E2 -627.991} C_VEL
LIN {X 0,Y 601.447,Z 320.562,A -85,B 0,C 180,E1 -630.67,E2 -630.67} C_VEL
LIN {X 0,Y 601.438,Z 320.571,A -85,B 0,C 180,E1 -633.35,E2 -633.35} C_VEL
LIN {X 0,Y 601.44,Z 320.563,A -85,B 0,C 180,E1 -636.037,E2 -636.037} C_VEL
LIN {X 0,Y 601.436,Z 320.572,A -85,B 0,C 180,E1 -638.738,E2 -638.738} C_VEL
LIN {X 0,Y 601.424,Z 320.565,A -85,B 0,C 180,E1 -641.458,E2 -641.458} C_VEL
LIN {X 0,Y 601.422,Z 320.571,A -85,B 0,C 180,E1 -644.206,E2 -644.206} C_VEL
LIN {X 0,Y 601.432,Z 320.565,A -85,B 0,C 180,E1 -646.986,E2 -646.986} C_VEL
LIN {X 0,Y 601.407,Z 320.569,A -85,B 0,C 180,E1 -649.81,E2 -649.81} C_VEL
LIN {X 0,Y 601.415,Z 320.571,A -85,B 0,C 180,E1 -652.683,E2 -652.683} C_VEL
LIN {X 0,Y 601.403,Z 320.573,A -85,B 0,C 180,E1 -654.879,E2 -654.879} C_VEL
LIN {X 0,Y 601.412,Z 320.567,A -85,B 0,C 180,E1 -657.362,E2 -657.362} C_VEL
LIN {X 0,Y 601.432,Z 320.57,A -85,B 0,C 180,E1 -660.149,E2 -660.149} C_VEL
LIN {X 0,Y 601.426,Z 320.565,A -85,B 0,C 180,E1 -662.716,E2 -662.716} C_VEL
LIN {X 0,Y 601.395,Z 320.574,A -85,B 0,C 180,E1 -665.112,E2 -665.112} C_VEL
LIN {X 0,Y 601.439,Z 320.566,A -85,B 0,C 180,E1 -667.419,E2 -667.419} C_VEL
LIN {X 0,Y 601.405,Z 320.568,A -85,B 0,C 180,E1 -669.996,E2 -669.996} C_VEL
LIN {X 0,Y 601.417,Z 320.57,A -85,B 0,C 180,E1 -672.67,E2 -672.67} C_VEL
LIN {X 0,Y 601.43,Z 320.567,A -85,B 0,C 180,E1 -675.482,E2 -675.482} C_VEL
LIN {X 0,Y 601.425,Z 320.565,A -85,B 0,C 180,E1 -678.407,E2 -678.407} C_VEL
LIN {X 0,Y 601.435,Z 320.567,A -85,B 0,C 180,E1 -681.529,E2 -681.529} C_VEL
LIN {X 0,Y 601.393,Z 320.57,A -85,B 0,C 180,E1 -684.246,E2 -684.246} C_VEL
LIN {X 0,Y 601.431,Z 320.57,A -85,B 0,C 180,E1 -686.687,E2 -686.687} C_VEL
LIN {X 0,Y 601.418,Z 320.566,A -85,B 0,C 180,E1 -689.058,E2 -689.058} C_VEL
LIN {X 0,Y 601.432,Z 320.566,A -85,B 0,C 180,E1 -691.373,E2 -691.373} C_VEL
LIN {X 0,Y 601.408,Z 320.575,A -85,B 0,C 180,E1 -693.637,E2 -693.637} C_VEL
LIN {X 0,Y 601.462,Z 320.562,A -85,B 0,C 180,E1 -695.86,E2 -695.86} C_VEL
LIN {X 0,Y 601.406,Z 320.573,A -85,B 0,C 180,E1 -698.761,E2 -698.761} C_VEL
LIN {X 0,Y 601.403,Z 320.568,A -85,B 0,C 180,E1 -701.608,E2 -701.608} C_VEL
LIN {X 0,Y 601.42,Z 320.571,A -85,B 0,C 180,E1 -704.409,E2 -704.409} C_VEL
LIN {X 0,Y 601.423,Z 320.566,A -85,B 0,C 180,E1 -707.172,E2 -707.172} C_VEL
LIN {X 0,Y 601.431,Z 320.567,A -85,B 0,C 180,E1 -709.905,E2 -709.905} C_VEL
LIN {X 0,Y 601.446,Z 320.564,A -85,B 0,C 180,E1 -712.615,E2 -712.615} C_VEL
LIN {X 0,Y 601.424,Z 320.567,A -85,B 0,C 180,E1 -715.308,E2 -715.308} C_VEL
LIN {X 0,Y 601.422,Z 320.568,A -85,B 0,C 180,E1 -717.991,E2 -717.991} C_VEL
LIN {X 0,Y 601.451,Z 320.563,A -85,B 0,C 180,E1 -720.67,E2 -720.67} C_VEL
LIN {X 0,Y 601.431,Z 320.568,A -85,B 0,C 180,E1 -723.35,E2 -723.35} C_VEL
LIN {X 0,Y 601.408,Z 320.568,A -85,B 0,C 180,E1 -726.037,E2 -726.037} C_VEL
LIN {X 0,Y 601.421,Z 320.57,A -85,B 0,C 180,E1 -728.738,E2 -728.738} C_VEL
LIN {X 0,Y 601.439,Z 320.564,A -85,B 0,C 180,E1 -731.458,E2 -731.458} C_VEL
LIN {X 0,Y 601.418,Z 320.573,A -85,B 0,C 180,E1 -734.206,E2 -734.206} C_VEL
LIN {X 0,Y 601.42,Z 320.565,A -85,B 0,C 180,E1 -736.986,E2 -736.986} C_VEL
LIN {X 0,Y 601.412,Z 320.572,A -85,B 0,C 180,E1 -739.809,E2 -739.809} C_VEL
LIN {X 0,Y 601.417,Z 320.568,A -85,B 0,C 180,E1 -742.683,E2 -742.683} C_VEL
LIN {X 0,Y 601.406,Z 320.575,A -85,B 0,C 180,E1 -744.879,E2 -744.879} C_VEL
LIN {X 0,Y 601.421,Z 320.566,A -85,B 0,C 180,E1 -747.362,E2 -747.362} C_VEL
LIN {X 0,Y 601.434,Z 320.571,A -85,B 0,C 180,E1 -750.164,E2 -750.164} C_VEL
LIN {X 0,Y 601.418,Z 320.566,A -85,B 0,C 180,E1 -752.714,E2 -752.714} C_VEL
LIN {X 0,Y 601.417,Z 320.568,A -85,B 0,C 180,E1 -755.114,E2 -755.114} C_VEL
LIN {X 0,Y 601.441,Z 320.57,A -85,B 0,C 180,E1 -757.419,E2 -757.419} C_VEL
LIN {X 0,Y 601.417,Z 320.566,A -85,B 0,C 180,E1 -759.995,E2 -759.995} C_VEL
LIN {X 0,Y 601.413,Z 320.575,A -85,B 0,C 180,E1 -762.67,E2 -762.67} C_VEL
LIN {X 0,Y 601.431,Z 320.565,A -85,B 0,C 180,E1 -765.482,E2 -765.482} C_VEL
LIN {X 0,Y 601.428,Z 320.567,A -85,B 0,C 180,E1 -768.407,E2 -768.407} C_VEL
LIN {X 0,Y 601.431,Z 320.573,A -85,B 0,C 180,E1 -771.53,E2 -771.53} C_VEL
LIN {X 0,Y 601.45,Z 320.726,A -85,B 0,C 180,E1 -774.115,E2 -774.115} C_VEL
LIN {X 0,Y 601.743,Z 325.508,A -85,B 0,C 180,E1 -775.089,E2 -775.089} C_VEL
LIN {X 0,Y 601.662,Z 340.829,A -85,B 0,C 180,E1 -778.091,E2 -778.091} C_VEL
LIN {X 0,Y 601.715,Z 352.19,A -85,B 0,C 180,E1 -780.238,E2 -780.238} C_VEL
LIN {X 0,Y 601.667,Z 365.885,A -85,B 0,C 180,E1 -782.899,E2 -782.899} C_VEL
LIN {X 0,Y 601.601,Z 379.338,A -85,B 0,C 180,E1 -785.453,E2 -785.453} C_VEL
LIN {X 0,Y 601.545,Z 393.275,A -85,B 0,C 180,E1 -788.046,E2 -788.046} C_VEL
LIN {X 0,Y 601.493,Z 408.926,A -85,B 0,C 180,E1 -790.903,E2 -790.903} C_VEL
LIN {X 0,Y 601.452,Z 424.578,A -85,B 0,C 180,E1 -793.713,E2 -793.713} C_VEL
LIN {X 0,Y 601.426,Z 440.229,A -85,B 0,C 180,E1 -796.484,E2 -796.484} C_VEL
LIN {X 0,Y 601.414,Z 449.156,A -85,B 0,C 180,E1 -798.05,E2 -798.05} C_VEL
LIN {X 0,Y 601.592,Z 461.433,A -85,B 0,C 180,E1 -798.267,E2 -798.267} C_VEL
LIN {X 0,Y 601.561,Z 474.224,A -85,B 0,C 180,E1 -798.622,E2 -798.622} C_VEL
LIN {X 0,Y 601.545,Z 485.884,A -85,B 0,C 180,E1 -799.073,E2 -799.073} C_VEL
LIN {X 0,Y 601.481,Z 497.325,A -85,B 0,C 180,E1 -799.651,E2 -799.651} C_VEL
LIN {X 0,Y 601.47,Z 507.929,A -85,B 0,C 180,E1 -800.33,E2 -800.33} C_VEL
LIN {X 0,Y 601.435,Z 517.597,A -85,B 0,C 180,E1 -801.093,E2 -801.093} C_VEL
LIN {X 0,Y 601.407,Z 526.412,A -85,B 0,C 180,E1 -801.939,E2 -801.939} C_VEL
LIN {X 0,Y 601.388,Z 533.69,A -85,B 0,C 180,E1 -802.783,E2 -802.783} C_VEL
LIN {X 0,Y 601.375,Z 540.773,A -85,B 0,C 180,E1 -803.782,E2 -803.782} C_VEL
LIN {X 0,Y 601.373,Z 545.68,A -85,B 0,C 180,E1 -804.635,E2 -804.635} C_VEL
LIN {X 0,Y 601.353,Z 550.371,A -85,B 0,C 180,E1 -805.643,E2 -805.643} C_VEL
LIN {X 0,Y 601.344,Z 553.956,A -85,B 0,C 180,E1 -806.65,E2 -806.65} C_VEL
LIN {X 0,Y 601.325,Z 555.809,A -85,B 0,C 180,E1 -807.32,E2 -807.32} C_VEL
LIN {X 0,Y 601.343,Z 557.201,A -85,B 0,C 180,E1 -807.991,E2 -807.991} C_VEL
LIN {X 0,Y 601.339,Z 558.784,A -85,B 0,C 180,E1 -809.33,E2 -809.33} C_VEL
LIN {X 0,Y 601.335,Z 559,A -85,B 0,C 180,E1 -810,E2 -810} C_VEL
LIN {X 0,Y 601.348,Z 558.184,A -85,B 0,C 180,E1 -811.339,E2 -811.339} C_VEL
LIN {X 0,Y 601.343,Z 557.202,A -85,B 0,C 180,E1 -812.009,E2 -812.009} C_VEL
LIN {X 0,Y 601.325,Z 555.809,A -85,B 0,C 180,E1 -812.68,E2 -812.68} C_VEL
LIN {X 0,Y 601.367,Z 552.896,A -85,B 0,C 180,E1 -813.685,E2 -813.685} C_VEL
LIN {X 0,Y 601.336,Z 548.95,A -85,B 0,C 180,E1 -814.693,E2 -814.693} C_VEL
LIN {X 0,Y 601.372,Z 542.877,A -85,B 0,C 180,E1 -815.869,E2 -815.869} C_VEL
LIN {X 0,Y 601.382,Z 536.235,A -85,B 0,C 180,E1 -816.88,E2 -816.88} C_VEL
LIN {X 0,Y 601.4,Z 527.989,A -85,B 0,C 180,E1 -817.892,E2 -817.892} C_VEL
LIN {X 0,Y 601.436,Z 519.536,A -85,B 0,C 180,E1 -818.738,E2 -818.738} C_VEL
LIN {X 0,Y 601.451,Z 509.091,A -85,B 0,C 180,E1 -819.585,E2 -819.585} C_VEL
LIN {X 0,Y 601.469,Z 498.756,A -85,B 0,C 180,E1 -820.265,E2 -820.265} C_VEL
LIN {X 0,Y 601.537,Z 486.602,A -85,B 0,C 180,E1 -820.896,E2 -820.896} C_VEL
LIN {X 0,Y 601.561,Z 474.217,A -85,B 0,C 180,E1 -821.379,E2 -821.379} C_VEL
LIN {X 0,Y 601.592,Z 461.435,A -85,B 0,C 180,E1 -821.733,E2 -821.733} C_VEL
LIN {X 0,Y 601.414,Z 449.156,A -85,B 0,C 180,E1 -821.95,E2 -821.95} C_VEL
LIN {X 0,Y 601.437,Z 432.404,A -85,B 0,C 180,E1 -824.897,E2 -824.897} C_VEL
LIN {X 0,Y 601.482,Z 416.753,A -85,B 0,C 180,E1 -827.686,E2 -827.686} C_VEL
LIN {X 0,Y 601.512,Z 403.058,A -85,B 0,C 180,E1 -830.162,E2 -830.162} C_VEL
LIN {X 0,Y 601.588,Z 387.406,A -85,B 0,C 180,E1 -833.039,E2 -833.039} C_VEL
LIN {X 0,Y 601.656,Z 371.212,A -85,B 0,C 180,E1 -836.082,E2 -836.082} C_VEL
LIN {X 0,Y 601.69,Z 356.939,A -85,B 0,C 180,E1 -838.832,E2 -838.832} C_VEL
LIN {X 0,Y 601.685,Z 346.993,A -85,B 0,C 180,E1 -840.732,E2 -840.732} C_VEL
LIN {X 0,Y 601.527,Z 328.539,A -85,B 0,C 180,E1 -843.949,E2 -843.949} C_VEL
LIN {X 0,Y 601.437,Z 320.569,A -85,B 0,C 180,E1 -845.408,E2 -845.408} C_VEL
LIN {X 0,Y 601.437,Z 320.569,A -85,B 0,C 180,E1 -848.471,E2 -848.471} C_VEL
LIN {X 0,Y 601.429,Z 320.573,A -85,B 0,C 180,E1 -851.593,E2 -851.593} C_VEL
LIN {X 0,Y 601.429,Z 320.572,A -85,B 0,C 180,E1 -854.535,E2 -854.535} C_VEL
LIN {X 0,Y 601.412,Z 320.574,A -85,B 0,C 180,E1 -857.41,E2 -857.41} C_VEL
LIN {X 0,Y 601.406,Z 320.575,A -85,B 0,C 180,E1 -860.004,E2 -860.004} C_VEL
LIN {X 0,Y 601.441,Z 320.568,A -85,B 0,C 180,E1 -862.618,E2 -862.618} C_VEL
LIN {X 0,Y 601.441,Z 320.566,A -85,B 0,C 180,E1 -865.07,E2 -865.07} C_VEL
LIN {X 0,Y 601.426,Z 320.569,A -85,B 0,C 180,E1 -867.484,E2 -867.484} C_VEL
LIN {X 0,Y 601.434,Z 320.572,A -85,B 0,C 180,E1 -869.852,E2 -869.852} C_VEL
LIN {X 0,Y 601.424,Z 320.572,A -85,B 0,C 180,E1 -872.637,E2 -872.637} C_VEL
LIN {X 0,Y 601.408,Z 320.571,A -85,B 0,C 180,E1 -875.122,E2 -875.122} C_VEL
LIN {X 0,Y 601.421,Z 320.57,A -85,B 0,C 180,E1 -877.395,E2 -877.395} C_VEL
LIN {X 0,Y 601.408,Z 320.571,A -85,B 0,C 180,E1 -880.191,E2 -880.191} C_VEL
LIN {X 0,Y 601.42,Z 320.57,A -85,B 0,C 180,E1 -883.014,E2 -883.014} C_VEL
LIN {X 0,Y 601.427,Z 320.569,A -85,B 0,C 180,E1 -885.908,E2 -885.908} C_VEL
LIN {X 0,Y 601.451,Z 320.565,A -85,B 0,C 180,E1 -887.537,E2 -887.537} C_VEL
LIN {X 0,Y 601.535,Z 333.875,A -85,B 0,C 180,E1 -888.031,E2 -888.031} C_VEL
LIN {X 0,Y 601.511,Z 346.028,A -85,B 0,C 180,E1 -888.625,E2 -888.625} C_VEL
LIN {X 0,Y 601.473,Z 357.027,A -85,B 0,C 180,E1 -889.31,E2 -889.31} C_VEL
LIN {X 0,Y 601.443,Z 366.878,A -85,B 0,C 180,E1 -890.075,E2 -890.075} C_VEL
LIN {X 0,Y 601.431,Z 375.831,A -85,B 0,C 180,E1 -890.923,E2 -890.923} C_VEL
LIN {X 0,Y 601.407,Z 384.565,A -85,B 0,C 180,E1 -891.939,E2 -891.939} C_VEL
LIN {X 0,Y 601.377,Z 391.533,A -85,B 0,C 180,E1 -892.951,E2 -892.951} C_VEL
LIN {X 0,Y 601.36,Z 397.108,A -85,B 0,C 180,E1 -893.962,E2 -893.962} C_VEL
LIN {X 0,Y 601.339,Z 401.485,A -85,B 0,C 180,E1 -894.971,E2 -894.971} C_VEL
LIN {X 0,Y 601.345,Z 404.792,A -85,B 0,C 180,E1 -895.979,E2 -895.979} C_VEL
LIN {X 0,Y 601.34,Z 406.433,A -85,B 0,C 180,E1 -896.65,E2 -896.65} C_VEL
LIN {X 0,Y 601.34,Z 408.509,A -85,B 0,C 180,E1 -897.991,E2 -897.991} C_VEL
LIN {X 0,Y 601.339,Z 408.94,A -85,B 0,C 180,E1 -899.33,E2 -899.33} C_VEL
LIN {X 0,Y 601.336,Z 408.586,A -85,B 0,C 180,E1 -900,E2 -900} C_VEL
LIN {X 0,Y 601.34,Z 407.831,A -85,B 0,C 180,E1 -900.67,E2 -900.67} C_VEL
LIN {X 0,Y 601.349,Z 406.648,A -85,B 0,C 180,E1 -901.339,E2 -901.339} C_VEL
LIN {X 0,Y 601.358,Z 404.118,A -85,B 0,C 180,E1 -902.344,E2 -902.344} C_VEL
LIN {X 0,Y 601.349,Z 400.593,A -85,B 0,C 180,E1 -903.35,E2 -903.35} C_VEL
LIN {X 0,Y 601.357,Z 395.97,A -85,B 0,C 180,E1 -904.357,E2 -904.357} C_VEL
LIN {X 0,Y 601.385,Z 388.988,A -85,B 0,C 180,E1 -905.533,E2 -905.533} C_VEL
LIN {X 0,Y 601.401,Z 380.737,A -85,B 0,C 180,E1 -906.626,E2 -906.626} C_VEL
LIN {X 0,Y 601.419,Z 371.962,A -85,B 0,C 180,E1 -907.554,E2 -907.554} C_VEL
LIN {X 0,Y 601.455,Z 362.185,A -85,B 0,C 180,E1 -908.399,E2 -908.399} C_VEL
LIN {X 0,Y 601.483,Z 351.228,A -85,B 0,C 180,E1 -909.16,E2 -909.16} C_VEL
LIN {X 0,Y 601.51,Z 338.782,A -85,B 0,C 180,E1 -909.839,E2 -909.839} C_VEL
LIN {X 0,Y 601.541,Z 331.55,A -85,B 0,C 180,E1 -910.157,E2 -910.157} C_VEL
LIN {X 0,Y 601.2,Z 328.414,A -85,B 0,C 180,E1 -910.348,E2 -910.348} C_VEL
LIN {X 0,Y 600.345,Z 325.984,A -85,B 0,C 180,E1 -910.613,E2 -910.613} C_VEL
LIN {X 0,Y 598.575,Z 323.501,A -85,B 0,C 180,E1 -911.091,E2 -911.091} C_VEL
LIN {X 0,Y 596.031,Z 321.9,A -85,B 0,C 180,E1 -911.834,E2 -911.834} C_VEL
LIN {X 0,Y 594.45,Z 321.456,A -85,B 0,C 180,E1 -912.631,E2 -912.631} C_VEL
LIN {X 0,Y 594.369,Z 321.444,A -85,B 0,C 180,E1 -912.835,E2 -912.835} C_VEL
LIN {X 0,Y 594.376,Z 321.445,A -85,B 0,C 180,E1 -915.078,E2 -915.078} C_VEL
LIN {X 0,Y 594.388,Z 321.448,A -85,B 0,C 180,E1 -917.193,E2 -917.193} C_VEL
LIN {X 0,Y 594.378,Z 321.443,A -85,B 0,C 180,E1 -920.054,E2 -920.054} C_VEL
LIN {X 0,Y 594.362,Z 321.448,A -85,B 0,C 180,E1 -922.967,E2 -922.967} C_VEL
LIN {X 0,Y 594.377,Z 321.443,A -85,B 0,C 180,E1 -925.193,E2 -925.193} C_VEL
LIN {X 0,Y 594.39,Z 321.444,A -85,B 0,C 180,E1 -927.526,E2 -927.526} C_VEL
LIN {X 0,Y 594.392,Z 321.442,A -85,B 0,C 180,E1 -930.328,E2 -930.328} C_VEL
LIN {X 0,Y 594.381,Z 321.446,A -85,B 0,C 180,E1 -932.95,E2 -932.95} C_VEL
LIN {X 0,Y 594.354,Z 321.448,A -85,B 0,C 180,E1 -935.409,E2 -935.409} C_VEL
LIN {X 0,Y 594.39,Z 321.442,A -85,B 0,C 180,E1 -937.94,E2 -937.94} C_VEL
LIN {X 0,Y 594.38,Z 321.444,A -85,B 0,C 180,E1 -940.822,E2 -940.822} C_VEL
LIN {X 0,Y 594.369,Z 321.445,A -85,B 0,C 180,E1 -943.299,E2 -943.299} C_VEL
LIN {X 0,Y 594.386,Z 321.444,A -85,B 0,C 180,E1 -946.159,E2 -946.159} C_VEL
LIN {X 0,Y 594.383,Z 321.451,A -85,B 0,C 180,E1 -949.177,E2 -949.177} C_VEL
LIN {X 0,Y 594.386,Z 321.442,A -85,B 0,C 180,E1 -952.059,E2 -952.059} C_VEL
LIN {X 0,Y 594.354,Z 321.451,A -85,B 0,C 180,E1 -954.676,E2 -954.676} C_VEL
LIN {X 0,Y 594.382,Z 321.442,A -85,B 0,C 180,E1 -957.088,E2 -957.088} C_VEL
LIN {X 0,Y 594.388,Z 321.448,A -85,B 0,C 180,E1 -959.672,E2 -959.672} C_VEL
LIN {X 0,Y 594.377,Z 321.443,A -85,B 0,C 180,E1 -962.539,E2 -962.539} C_VEL
LIN {X 0,Y 594.38,Z 321.447,A -85,B 0,C 180,E1 -964.807,E2 -964.807} C_VEL
LIN {X 0,Y 594.368,Z 321.447,A -85,B 0,C 180,E1 -967.264,E2 -967.264} C_VEL
LIN {X 0,Y 594.374,Z 321.445,A -85,B 0,C 180,E1 -969.946,E2 -969.946} C_VEL
LIN {X 0,Y 594.389,Z 321.442,A -85,B 0,C 180,E1 -972.807,E2 -972.807} C_VEL
LIN {X 0,Y 594.392,Z 321.448,A -85,B 0,C 180,E1 -975.826,E2 -975.826} C_VEL
LIN {X 0,Y 594.388,Z 321.442,A -85,B 0,C 180,E1 -978.404,E2 -978.404} C_VEL
LIN {X 0,Y 594.381,Z 321.449,A -85,B 0,C 180,E1 -981.158,E2 -981.158} C_VEL
LIN {X 0,Y 594.389,Z 321.442,A -85,B 0,C 180,E1 -983.891,E2 -983.891} C_VEL
LIN {X 0,Y 594.379,Z 321.447,A -85,B 0,C 180,E1 -986.611,E2 -986.611} C_VEL
LIN {X 0,Y 594.419,Z 321.439,A -85,B 0,C 180,E1 -989.323,E2 -989.323} C_VEL
LIN {X 0,Y 594.406,Z 321.442,A -85,B 0,C 180,E1 -992.033,E2 -992.033} C_VEL
LIN {X 0,Y 594.388,Z 321.444,A -85,B 0,C 180,E1 -994.748,E2 -994.748} C_VEL
LIN {X 0,Y 594.396,Z 321.442,A -85,B 0,C 180,E1 -997.473,E2 -997.473} C_VEL
LIN {X 0,Y 594.402,Z 321.444,A -85,B 0,C 180,E1 -1000.216,E2 -1000.216} C_VEL
LIN {X 0,Y 594.369,Z 321.444,A -85,B 0,C 180,E1 -1002.983,E2 -1002.983} C_VEL
LIN {X 0,Y 594.371,Z 321.444,A -85,B 0,C 180,E1 -1005.078,E2 -1005.078} C_VEL
LIN {X 0,Y 594.389,Z 321.444,A -85,B 0,C 180,E1 -1007.194,E2 -1007.194} C_VEL
LIN {X 0,Y 594.376,Z 321.444,A -85,B 0,C 180,E1 -1010.054,E2 -1010.054} C_VEL
LIN {X 0,Y 594.367,Z 321.452,A -85,B 0,C 180,E1 -1012.967,E2 -1012.967} C_VEL
LIN {X 0,Y 594.378,Z 321.444,A -85,B 0,C 180,E1 -1015.193,E2 -1015.193} C_VEL
LIN {X 0,Y 594.388,Z 321.442,A -85,B 0,C 180,E1 -1017.527,E2 -1017.527} C_VEL
LIN {X 0,Y 594.389,Z 321.445,A -85,B 0,C 180,E1 -1020.328,E2 -1020.328} C_VEL
LIN {X 0,Y 594.382,Z 321.443,A -85,B 0,C 180,E1 -1022.95,E2 -1022.95} C_VEL
LIN {X 0,Y 594.351,Z 321.453,A -85,B 0,C 180,E1 -1025.409,E2 -1025.409} C_VEL
LIN {X 0,Y 594.388,Z 321.442,A -85,B 0,C 180,E1 -1027.941,E2 -1027.941} C_VEL
LIN {X 0,Y 594.381,Z 321.448,A -85,B 0,C 180,E1 -1030.822,E2 -1030.822} C_VEL
LIN {X 0,Y 594.387,Z 321.446,A -85,B 0,C 180,E1 -1033.841,E2 -1033.841} C_VEL
LIN {X 0,Y 594.37,Z 321.444,A -85,B 0,C 180,E1 -1036.701,E2 -1036.701} C_VEL
LIN {X 0,Y 594.371,Z 321.452,A -85,B 0,C 180,E1 -1039.433,E2 -1039.433} C_VEL
LIN {X 0,Y 594.392,Z 321.442,A -85,B 0,C 180,E1 -1042.392,E2 -1042.392} C_VEL
LIN {X 0,Y 594.398,Z 321.441,A -85,B 0,C 180,E1 -1045.421,E2 -1045.421} C_VEL
LIN {X 0,Y 594.381,Z 321.45,A -85,B 0,C 180,E1 -1048.358,E2 -1048.358} C_VEL
LIN {X 0,Y 594.387,Z 321.442,A -85,B 0,C 180,E1 -1051.043,E2 -1051.043} C_VEL
LIN {X 0,Y 594.386,Z 321.445,A -85,B 0,C 180,E1 -1053.979,E2 -1053.979} C_VEL
LIN {X 0,Y 594.38,Z 321.443,A -85,B 0,C 180,E1 -1056.296,E2 -1056.296} C_VEL
LIN {X 0,Y 594.402,Z 321.443,A -85,B 0,C 180,E1 -1059.224,E2 -1059.224} C_VEL
LIN {X 0,Y 594.352,Z 321.449,A -85,B 0,C 180,E1 -1062.095,E2 -1062.095} C_VEL
LIN {X 0,Y 594.373,Z 321.452,A -85,B 0,C 180,E1 -1064.219,E2 -1064.219} C_VEL
LIN {X 0,Y 594.39,Z 321.445,A -85,B 0,C 180,E1 -1066.321,E2 -1066.321} C_VEL
LIN {X 0,Y 594.381,Z 321.445,A -85,B 0,C 180,E1 -1069.095,E2 -1069.095} C_VEL
LIN {X 0,Y 594.418,Z 321.439,A -85,B 0,C 180,E1 -1071.843,E2 -1071.843} C_VEL
LIN {X 0,Y 594.398,Z 321.445,A -85,B 0,C 180,E1 -1074.572,E2 -1074.572} C_VEL
LIN {X 0,Y 594.411,Z 321.439,A -85,B 0,C 180,E1 -1077.289,E2 -1077.289} C_VEL
LIN {X 0,Y 594.421,Z 321.443,A -85,B 0,C 180,E1 -1080,E2 -1080} C_VEL
LIN {X 0,Y 594.411,Z 321.439,A -85,B 0,C 180,E1 -1082.711,E2 -1082.711} C_VEL
LIN {X 0,Y 594.393,Z 321.449,A -85,B 0,C 180,E1 -1085.428,E2 -1085.428} C_VEL
LIN {X 0,Y 594.386,Z 321.442,A -85,B 0,C 180,E1 -1088.157,E2 -1088.157} C_VEL
LIN {X 0,Y 594.4,Z 321.444,A -85,B 0,C 180,E1 -1091.075,E2 -1091.075} C_VEL
LIN {X 0,Y 594.38,Z 321.443,A -85,B 0,C 180,E1 -1093.679,E2 -1093.679} C_VEL
LIN {X 0,Y 594.401,Z 321.443,A -85,B 0,C 180,E1 -1096.485,E2 -1096.485} C_VEL
LIN {X 0,Y 594.374,Z 321.447,A -85,B 0,C 180,E1 -1099.334,E2 -1099.334} C_VEL
LIN {X 0,Y 594.371,Z 321.451,A -85,B 0,C 180,E1 -1101.503,E2 -1101.503} C_VEL
LIN {X 0,Y 594.395,Z 321.443,A -85,B 0,C 180,E1 -1104.446,E2 -1104.446} C_VEL
LIN {X 0,Y 594.39,Z 321.45,A -85,B 0,C 180,E1 -1106.699,E2 -1106.699} C_VEL
LIN {X 0,Y 594.387,Z 321.443,A -85,B 0,C 180,E1 -1108.998,E2 -1108.998} C_VEL
LIN {X 0,Y 594.38,Z 321.445,A -85,B 0,C 180,E1 -1111.642,E2 -1111.642} C_VEL
LIN {X 0,Y 594.399,Z 321.44,A -85,B 0,C 180,E1 -1114.579,E2 -1114.579} C_VEL
LIN {X 0,Y 594.395,Z 321.445,A -85,B 0,C 180,E1 -1117.608,E2 -1117.608} C_VEL
LIN {X 0,Y 594.37,Z 321.448,A -85,B 0,C 180,E1 -1120.567,E2 -1120.567} C_VEL
LIN {X 0,Y 594.37,Z 321.444,A -85,B 0,C 180,E1 -1123.299,E2 -1123.299} C_VEL
LIN {X 0,Y 594.389,Z 321.45,A -85,B 0,C 180,E1 -1126.159,E2 -1126.159} C_VEL
LIN {X 0,Y 594.379,Z 321.444,A -85,B 0,C 180,E1 -1129.178,E2 -1129.178} C_VEL
LIN {X 0,Y 594.387,Z 321.445,A -85,B 0,C 180,E1 -1132.059,E2 -1132.059} C_VEL
LIN {X 0,Y 594.375,Z 321.514,A -85,B 0,C 180,E1 -1133.862,E2 -1133.862} C_VEL
LIN {X 0,Y 594.89,Z 326.132,A -85,B 0,C 180,E1 -1134.835,E2 -1134.835} C_VEL
LIN {X 0,Y 594.726,Z 340.339,A -85,B 0,C 180,E1 -1137.674,E2 -1137.674} C_VEL
LIN {X 0,Y 594.808,Z 354.949,A -85,B 0,C 180,E1 -1140.442,E2 -1140.442} C_VEL
LIN {X 0,Y 594.728,Z 369.798,A -85,B 0,C 180,E1 -1143.317,E2 -1143.317} C_VEL
LIN {X 0,Y 594.643,Z 383.493,A -85,B 0,C 180,E1 -1145.936,E2 -1145.936} C_VEL
LIN {X 0,Y 594.556,Z 397.188,A -85,B 0,C 180,E1 -1148.504,E2 -1148.504} C_VEL
LIN {X 0,Y 594.496,Z 412.839,A -85,B 0,C 180,E1 -1151.386,E2 -1151.386} C_VEL
LIN {X 0,Y 594.406,Z 428.491,A -85,B 0,C 180,E1 -1154.22,E2 -1154.22} C_VEL
LIN {X 0,Y 594.365,Z 442.186,A -85,B 0,C 180,E1 -1156.669,E2 -1156.669} C_VEL
LIN {X 0,Y 594.358,Z 449.156,A -85,B 0,C 180,E1 -1157.906,E2 -1157.906} C_VEL
LIN {X 0,Y 594.674,Z 454.938,A -85,B 0,C 180,E1 -1157.999,E2 -1157.999} C_VEL
LIN {X 0,Y 594.603,Z 468.212,A -85,B 0,C 180,E1 -1158.3,E2 -1158.3} C_VEL
LIN {X 0,Y 594.564,Z 481.216,A -85,B 0,C 180,E1 -1158.743,E2 -1158.743} C_VEL
LIN {X 0,Y 594.535,Z 492.63,A -85,B 0,C 180,E1 -1159.27,E2 -1159.27} C_VEL
LIN {X 0,Y 594.48,Z 504.198,A -85,B 0,C 180,E1 -1159.958,E2 -1159.958} C_VEL
LIN {X 0,Y 594.414,Z 514.594,A -85,B 0,C 180,E1 -1160.729,E2 -1160.729} C_VEL
LIN {X 0,Y 594.383,Z 523.111,A -85,B 0,C 180,E1 -1161.5,E2 -1161.5} C_VEL
LIN {X 0,Y 594.347,Z 530.959,A -85,B 0,C 180,E1 -1162.355,E2 -1162.355} C_VEL
LIN {X 0,Y 594.283,Z 538.812,A -85,B 0,C 180,E1 -1163.408,E2 -1163.408} C_VEL
LIN {X 0,Y 594.289,Z 545.68,A -85,B 0,C 180,E1 -1164.571,E2 -1164.571} C_VEL
LIN {X 0,Y 594.27,Z 550.371,A -85,B 0,C 180,E1 -1165.591,E2 -1165.591} C_VEL
LIN {X 0,Y 594.267,Z 553.956,A -85,B 0,C 180,E1 -1166.61,E2 -1166.61} C_VEL
LIN {X 0,Y 594.226,Z 555.809,A -85,B 0,C 180,E1 -1167.288,E2 -1167.288} C_VEL
LIN {X 0,Y 594.242,Z 557.201,A -85,B 0,C 180,E1 -1167.967,E2 -1167.967} C_VEL
LIN {X 0,Y 594.239,Z 558.784,A -85,B 0,C 180,E1 -1169.322,E2 -1169.322} C_VEL
LIN {X 0,Y 594.236,Z 559,A -85,B 0,C 180,E1 -1170,E2 -1170} C_VEL
LIN {X 0,Y 594.248,Z 558.185,A -85,B 0,C 180,E1 -1171.355,E2 -1171.355} C_VEL
LIN {X 0,Y 594.242,Z 557.202,A -85,B 0,C 180,E1 -1172.033,E2 -1172.033} C_VEL
LIN {X 0,Y 594.226,Z 555.81,A -85,B 0,C 180,E1 -1172.712,E2 -1172.712} C_VEL
LIN {X 0,Y 594.288,Z 552.896,A -85,B 0,C 180,E1 -1173.729,E2 -1173.729} C_VEL
LIN {X 0,Y 594.241,Z 548.95,A -85,B 0,C 180,E1 -1174.749,E2 -1174.749} C_VEL
LIN {X 0,Y 594.304,Z 542.877,A -85,B 0,C 180,E1 -1175.939,E2 -1175.939} C_VEL
LIN {X 0,Y 594.308,Z 536.236,A -85,B 0,C 180,E1 -1176.962,E2 -1176.962} C_VEL
LIN {X 0,Y 594.359,Z 527.989,A -85,B 0,C 180,E1 -1177.986,E2 -1177.986} C_VEL
LIN {X 0,Y 594.382,Z 519.537,A -85,B 0,C 180,E1 -1178.842,E2 -1178.842} C_VEL
LIN {X 0,Y 594.435,Z 509.093,A -85,B 0,C 180,E1 -1179.699,E2 -1179.699} C_VEL
LIN {X 0,Y 594.482,Z 498.758,A -85,B 0,C 180,E1 -1180.386,E2 -1180.386} C_VEL
LIN {X 0,Y 594.556,Z 487.741,A -85,B 0,C 180,E1 -1180.972,E2 -1180.972} C_VEL
LIN {X 0,Y 594.582,Z 475.715,A -85,B 0,C 180,E1 -1181.464,E2 -1181.464} C_VEL
LIN {X 0,Y 594.63,Z 462.349,A -85,B 0,C 180,E1 -1181.85,E2 -1181.85} C_VEL
LIN {X 0,Y 594.579,Z 450.597,A -85,B 0,C 180,E1 -1182.068,E2 -1182.068} C_VEL
LIN {X 0,Y 594.363,Z 449.034,A -85,B 0,C 180,E1 -1182.116,E2 -1182.116} C_VEL
LIN {X 0,Y 594.396,Z 434.361,A -85,B 0,C 180,E1 -1184.727,E2 -1184.727} C_VEL
LIN {X 0,Y 594.457,Z 418.709,A -85,B 0,C 180,E1 -1187.546,E2 -1187.546} C_VEL
LIN {X 0,Y 594.533,Z 405.014,A -85,B 0,C 180,E1 -1190.048,E2 -1190.048} C_VEL
LIN {X 0,Y 594.623,Z 389.363,A -85,B 0,C 180,E1 -1192.957,E2 -1192.957} C_VEL
LIN {X 0,Y 594.706,Z 373.711,A -85,B 0,C 180,E1 -1195.929,E2 -1195.929} C_VEL
LIN {X 0,Y 594.786,Z 360.016,A -85,B 0,C 180,E1 -1198.591,E2 -1198.591} C_VEL
LIN {X 0,Y 594.739,Z 351.899,A -85,B 0,C 180,E1 -1200.069,E2 -1200.069} C_VEL
LIN {X 0,Y 594.516,Z 334.366,A -85,B 0,C 180,E1 -1203.144,E2 -1203.144} C_VEL
LIN {X 0,Y 594.479,Z 321.969,A -85,B 0,C 180,E1 -1205.4,E2 -1205.4} C_VEL
LIN {X 0,Y 594.402,Z 321.446,A -85,B 0,C 180,E1 -1205.51,E2 -1205.51} C_VEL
LIN {X 0,Y 594.388,Z 321.446,A -85,B 0,C 180,E1 -1207.941,E2 -1207.941} C_VEL
LIN {X 0,Y 594.378,Z 321.447,A -85,B 0,C 180,E1 -1210.822,E2 -1210.822} C_VEL
LIN {X 0,Y 594.372,Z 321.449,A -85,B 0,C 180,E1 -1213.299,E2 -1213.299} C_VEL
LIN {X 0,Y 594.372,Z 321.449,A -85,B 0,C 180,E1 -1216.161,E2 -1216.161} C_VEL
LIN {X 0,Y 594.382,Z 321.446,A -85,B 0,C 180,E1 -1219.178,E2 -1219.178} C_VEL
LIN {X 0,Y 594.391,Z 321.444,A -85,B 0,C 180,E1 -1222.059,E2 -1222.059} C_VEL
LIN {X 0,Y 594.365,Z 321.449,A -85,B 0,C 180,E1 -1224.675,E2 -1224.675} C_VEL
LIN {X 0,Y 594.381,Z 321.451,A -85,B 0,C 180,E1 -1227.089,E2 -1227.089} C_VEL
LIN {X 0,Y 594.393,Z 321.446,A -85,B 0,C 180,E1 -1229.672,E2 -1229.672} C_VEL
LIN {X 0,Y 594.38,Z 321.448,A -85,B 0,C 180,E1 -1232.539,E2 -1232.539} C_VEL
LIN {X 0,Y 594.379,Z 321.446,A -85,B 0,C 180,E1 -1234.807,E2 -1234.807} C_VEL
LIN {X 0,Y 594.367,Z 321.449,A -85,B 0,C 180,E1 -1237.265,E2 -1237.265} C_VEL
LIN {X 0,Y 594.376,Z 321.45,A -85,B 0,C 180,E1 -1239.946,E2 -1239.946} C_VEL
LIN {X 0,Y 594.385,Z 321.448,A -85,B 0,C 180,E1 -1242.806,E2 -1242.806} C_VEL
LIN {X 0,Y 594.395,Z 321.445,A -85,B 0,C 180,E1 -1245.826,E2 -1245.826} C_VEL
LIN {X 0,Y 594.427,Z 321.441,A -85,B 0,C 180,E1 -1247.431,E2 -1247.431} C_VEL
LIN {X 0,Y 594.575,Z 333.614,A -85,B 0,C 180,E1 -1247.889,E2 -1247.889} C_VEL
LIN {X 0,Y 594.518,Z 345.963,A -85,B 0,C 180,E1 -1248.497,E2 -1248.497} C_VEL
LIN {X 0,Y 594.47,Z 356.862,A -85,B 0,C 180,E1 -1249.183,E2 -1249.183} C_VEL
LIN {X 0,Y 594.401,Z 366.747,A -85,B 0,C 180,E1 -1249.956,E2 -1249.956} C_VEL
LIN {X 0,Y 594.367,Z 375.723,A -85,B 0,C 180,E1 -1250.815,E2 -1250.815} C_VEL
LIN {X 0,Y 594.326,Z 384.477,A -85,B 0,C 180,E1 -1251.842,E2 -1251.842} C_VEL
LIN {X 0,Y 594.306,Z 391.467,A -85,B 0,C 180,E1 -1252.867,E2 -1252.867} C_VEL
LIN {X 0,Y 594.282,Z 397.056,A -85,B 0,C 180,E1 -1253.89,E2 -1253.89} C_VEL
LIN {X 0,Y 594.246,Z 401.446,A -85,B 0,C 180,E1 -1254.911,E2 -1254.911} C_VEL
LIN {X 0,Y 594.262,Z 404.765,A -85,B 0,C 180,E1 -1255.931,E2 -1255.931} C_VEL
LIN {X 0,Y 594.26,Z 406.41,A -85,B 0,C 180,E1 -1256.61,E2 -1256.61} C_VEL
LIN {X 0,Y 594.239,Z 408.498,A -85,B 0,C 180,E1 -1257.967,E2 -1257.967} C_VEL
LIN {X 0,Y 594.249,Z 408.915,A -85,B 0,C 180,E1 -1258.645,E2 -1258.645} C_VEL
LIN {X 0,Y 594.237,Z 408.594,A -85,B 0,C 180,E1 -1260,E2 -1260} C_VEL
LIN {X 0,Y 594.24,Z 407.848,A -85,B 0,C 180,E1 -1260.678,E2 -1260.678} C_VEL
LIN {X 0,Y 594.249,Z 406.673,A -85,B 0,C 180,E1 -1261.355,E2 -1261.355} C_VEL
LIN {X 0,Y 594.247,Z 405.093,A -85,B 0,C 180,E1 -1262.033,E2 -1262.033} C_VEL
LIN {X 0,Y 594.278,Z 401.912,A -85,B 0,C 180,E1 -1263.05,E2 -1263.05} C_VEL
LIN {X 0,Y 594.262,Z 397.679,A -85,B 0,C 180,E1 -1264.069,E2 -1264.069} C_VEL
LIN {X 0,Y 594.277,Z 391.254,A -85,B 0,C 180,E1 -1265.259,E2 -1265.259} C_VEL
LIN {X 0,Y 594.311,Z 384.4,A -85,B 0,C 180,E1 -1266.259,E2 -1266.259} C_VEL
LIN {X 0,Y 594.359,Z 375.465,A -85,B 0,C 180,E1 -1267.303,E2 -1267.303} C_VEL
LIN {X 0,Y 594.421,Z 365.497,A -85,B 0,C 180,E1 -1268.242,E2 -1268.242} C_VEL
LIN {X 0,Y 594.458,Z 355.317,A -85,B 0,C 180,E1 -1269.012,E2 -1269.012} C_VEL
LIN {X 0,Y 594.51,Z 344.055,A -85,B 0,C 180,E1 -1269.698,E2 -1269.698} C_VEL
LIN {X 0,Y 594.579,Z 332.075,A -85,B 0,C 180,E1 -1270.267,E2 -1270.267} C_VEL
LIN {X 0,Y 594.446,Z 321.718,A -85,B 0,C 180,E1 -1270.645,E2 -1270.645} C_VEL
LIN {X 0,Y 594.389,Z 321.444,A -85,B 0,C 180,E1 -1270.733,E2 -1270.733} C_VEL
LIN {X 0,Y 594.369,Z 321.444,A -85,B 0,C 180,E1 -1272.835,E2 -1272.835} C_VEL
LIN {X 0,Y 593.706,Z 321.531,A -85,B 0,C 180,E1 -1273.4,E2 -1273.4} C_VEL
LIN {X 0,Y 590.841,Z 321.885,A -85,B 0,C 180,E1 -1274.318,E2 -1274.318} C_VEL
LIN {X 0,Y 588.425,Z 322.186,A -85,B 0,C 180,E1 -1275.056,E2 -1275.056} C_VEL
LIN {X 0,Y 587.399,Z 322.32,A -85,B 0,C 180,E1 -1275.626,E2 -1275.626} C_VEL
LIN {X 0,Y 587.322,Z 322.324,A -85,B 0,C 180,E1 -1275.819,E2 -1275.819} C_VEL
LIN {X 0,Y 587.304,Z 322.324,A -85,B 0,C 180,E1 -1278.127,E2 -1278.127} C_VEL
LIN {X 0,Y 587.336,Z 322.326,A -85,B 0,C 180,E1 -1281.037,E2 -1281.037} C_VEL
LIN {X 0,Y 587.32,Z 322.323,A -85,B 0,C 180,E1 -1283.259,E2 -1283.259} C_VEL
LIN {X 0,Y 587.334,Z 322.321,A -85,B 0,C 180,E1 -1285.517,E2 -1285.517} C_VEL
LIN {X 0,Y 587.352,Z 322.325,A -85,B 0,C 180,E1 -1287.817,E2 -1287.817} C_VEL
LIN {X 0,Y 587.347,Z 322.319,A -85,B 0,C 180,E1 -1290.511,E2 -1290.511} C_VEL
LIN {X 0,Y 587.338,Z 322.326,A -85,B 0,C 180,E1 -1293.396,E2 -1293.396} C_VEL
LIN {X 0,Y 587.295,Z 322.325,A -85,B 0,C 180,E1 -1295.9,E2 -1295.9} C_VEL
LIN {X 0,Y 587.336,Z 322.327,A -85,B 0,C 180,E1 -1298.479,E2 -1298.479} C_VEL
LIN {X 0,Y 587.339,Z 322.32,A -85,B 0,C 180,E1 -1301.157,E2 -1301.157} C_VEL
LIN {X 0,Y 587.33,Z 322.326,A -85,B 0,C 180,E1 -1304.113,E2 -1304.113} C_VEL
LIN {X 0,Y 587.326,Z 322.324,A -85,B 0,C 180,E1 -1306.994,E2 -1306.994} C_VEL
LIN {X 0,Y 587.316,Z 322.324,A -85,B 0,C 180,E1 -1309.745,E2 -1309.745} C_VEL
LIN {X 0,Y 587.346,Z 322.322,A -85,B 0,C 180,E1 -1312.392,E2 -1312.392} C_VEL
LIN {X 0,Y 587.364,Z 322.318,A -85,B 0,C 180,E1 -1315.78,E2 -1315.78} C_VEL
LIN {X 0,Y 587.346,Z 322.324,A -85,B 0,C 180,E1 -1318.231,E2 -1318.231} C_VEL
LIN {X 0,Y 587.353,Z 322.319,A -85,B 0,C 180,E1 -1320.866,E2 -1320.866} C_VEL
LIN {X 0,Y 587.362,Z 322.319,A -85,B 0,C 180,E1 -1323.819,E2 -1323.819} C_VEL
LIN {X 0,Y 587.337,Z 322.32,A -85,B 0,C 180,E1 -1325.993,E2 -1325.993} C_VEL
LIN {X 0,Y 587.326,Z 322.324,A -85,B 0,C 180,E1 -1328.226,E2 -1328.226} C_VEL
LIN {X 0,Y 587.351,Z 322.318,A -85,B 0,C 180,E1 -1331.151,E2 -1331.151} C_VEL
LIN {X 0,Y 587.329,Z 322.329,A -85,B 0,C 180,E1 -1334.025,E2 -1334.025} C_VEL
LIN {X 0,Y 587.361,Z 322.32,A -85,B 0,C 180,E1 -1336.154,E2 -1336.154} C_VEL
LIN {X 0,Y 587.344,Z 322.323,A -85,B 0,C 180,E1 -1338.962,E2 -1338.962} C_VEL
LIN {X 0,Y 587.366,Z 322.317,A -85,B 0,C 180,E1 -1341.745,E2 -1341.745} C_VEL
LIN {X 0,Y 587.37,Z 322.323,A -85,B 0,C 180,E1 -1344.507,E2 -1344.507} C_VEL
LIN {X 0,Y 587.371,Z 322.316,A -85,B 0,C 180,E1 -1347.257,E2 -1347.257} C_VEL
LIN {X 0,Y 587.386,Z 322.321,A -85,B 0,C 180,E1 -1350,E2 -1350} C_VEL
LIN {X 0,Y 587.373,Z 322.316,A -85,B 0,C 180,E1 -1352.743,E2 -1352.743} C_VEL
LIN {X 0,Y 587.37,Z 322.32,A -85,B 0,C 180,E1 -1355.493,E2 -1355.493} C_VEL
LIN {X 0,Y 587.372,Z 322.318,A -85,B 0,C 180,E1 -1358.255,E2 -1358.255} C_VEL
LIN {X 0,Y 587.35,Z 322.319,A -85,B 0,C 180,E1 -1361.134,E2 -1361.134} C_VEL
LIN {X 0,Y 587.367,Z 322.321,A -85,B 0,C 180,E1 -1364.261,E2 -1364.261} C_VEL
LIN {X 0,Y 587.35,Z 322.324,A -85,B 0,C 180,E1 -1367.406,E2 -1367.406} C_VEL
LIN {X 0,Y 587.332,Z 322.321,A -85,B 0,C 180,E1 -1370.305,E2 -1370.305} C_VEL
LIN {X 0,Y 587.324,Z 322.325,A -85,B 0,C 180,E1 -1373.259,E2 -1373.259} C_VEL
LIN {X 0,Y 587.338,Z 322.32,A -85,B 0,C 180,E1 -1375.517,E2 -1375.517} C_VEL
LIN {X 0,Y 587.35,Z 322.321,A -85,B 0,C 180,E1 -1377.818,E2 -1377.818} C_VEL
LIN {X 0,Y 587.339,Z 322.321,A -85,B 0,C 180,E1 -1380.51,E2 -1380.51} C_VEL
LIN {X 0,Y 587.339,Z 322.326,A -85,B 0,C 180,E1 -1383.397,E2 -1383.397} C_VEL
LIN {X 0,Y 587.294,Z 322.326,A -85,B 0,C 180,E1 -1385.9,E2 -1385.9} C_VEL
LIN {X 0,Y 587.332,Z 322.324,A -85,B 0,C 180,E1 -1388.48,E2 -1388.48} C_VEL
LIN {X 0,Y 587.339,Z 322.321,A -85,B 0,C 180,E1 -1391.157,E2 -1391.157} C_VEL
LIN {X 0,Y 587.339,Z 322.328,A -85,B 0,C 180,E1 -1394.115,E2 -1394.115} C_VEL
LIN {X 0,Y 587.319,Z 322.323,A -85,B 0,C 180,E1 -1396.994,E2 -1396.994} C_VEL
LIN {X 0,Y 587.316,Z 322.326,A -85,B 0,C 180,E1 -1399.746,E2 -1399.746} C_VEL
LIN {X 0,Y 587.347,Z 322.319,A -85,B 0,C 180,E1 -1402.393,E2 -1402.393} C_VEL
LIN {X 0,Y 587.37,Z 322.316,A -85,B 0,C 180,E1 -1405.781,E2 -1405.781} C_VEL
LIN {X 0,Y 587.343,Z 322.327,A -85,B 0,C 180,E1 -1408.231,E2 -1408.231} C_VEL
LIN {X 0,Y 587.354,Z 322.318,A -85,B 0,C 180,E1 -1410.867,E2 -1410.867} C_VEL
LIN {X 0,Y 587.362,Z 322.322,A -85,B 0,C 180,E1 -1413.82,E2 -1413.82} C_VEL
LIN {X 0,Y 587.334,Z 322.321,A -85,B 0,C 180,E1 -1415.993,E2 -1415.993} C_VEL
LIN {X 0,Y 587.323,Z 322.322,A -85,B 0,C 180,E1 -1418.226,E2 -1418.226} C_VEL
LIN {X 0,Y 587.349,Z 322.32,A -85,B 0,C 180,E1 -1421.151,E2 -1421.151} C_VEL
LIN {X 0,Y 587.327,Z 322.326,A -85,B 0,C 180,E1 -1424.025,E2 -1424.025} C_VEL
LIN {X 0,Y 587.367,Z 322.322,A -85,B 0,C 180,E1 -1426.155,E2 -1426.155} C_VEL
LIN {X 0,Y 587.347,Z 322.32,A -85,B 0,C 180,E1 -1428.963,E2 -1428.963} C_VEL
LIN {X 0,Y 587.373,Z 322.318,A -85,B 0,C 180,E1 -1431.745,E2 -1431.745} C_VEL
LIN {X 0,Y 587.362,Z 322.32,A -85,B 0,C 180,E1 -1434.507,E2 -1434.507} C_VEL
LIN {X 0,Y 587.377,Z 322.315,A -85,B 0,C 180,E1 -1437.257,E2 -1437.257} C_VEL
LIN {X 0,Y 587.39,Z 322.319,A -85,B 0,C 180,E1 -1440,E2 -1440} C_VEL
LIN {X 0,Y 587.378,Z 322.315,A -85,B 0,C 180,E1 -1442.743,E2 -1442.743} C_VEL
LIN {X 0,Y 587.358,Z 322.325,A -85,B 0,C 180,E1 -1445.493,E2 -1445.493} C_VEL
LIN {X 0,Y 587.347,Z 322.319,A -85,B 0,C 180,E1 -1448.256,E2 -1448.256} C_VEL
LIN {X 0,Y 587.356,Z 322.321,A -85,B 0,C 180,E1 -1451.134,E2 -1451.134} C_VEL
LIN {X 0,Y 587.364,Z 322.324,A -85,B 0,C 180,E1 -1454.257,E2 -1454.257} C_VEL
LIN {X 0,Y 587.358,Z 322.319,A -85,B 0,C 180,E1 -1457.406,E2 -1457.406} C_VEL
LIN {X 0,Y 587.331,Z 322.321,A -85,B 0,C 180,E1 -1460.305,E2 -1460.305} C_VEL
LIN {X 0,Y 587.319,Z 322.329,A -85,B 0,C 180,E1 -1463.259,E2 -1463.259} C_VEL
LIN {X 0,Y 587.335,Z 322.322,A -85,B 0,C 180,E1 -1465.517,E2 -1465.517} C_VEL
LIN {X 0,Y 587.354,Z 322.319,A -85,B 0,C 180,E1 -1467.818,E2 -1467.818} C_VEL
LIN {X 0,Y 587.342,Z 322.324,A -85,B 0,C 180,E1 -1470.51,E2 -1470.51} C_VEL
LIN {X 0,Y 587.338,Z 322.322,A -85,B 0,C 180,E1 -1473.397,E2 -1473.397} C_VEL
LIN {X 0,Y 587.3,Z 322.328,A -85,B 0,C 180,E1 -1475.9,E2 -1475.9} C_VEL
LIN {X 0,Y 587.337,Z 322.321,A -85,B 0,C 180,E1 -1478.479,E2 -1478.479} C_VEL
LIN {X 0,Y 587.339,Z 322.324,A -85,B 0,C 180,E1 -1481.157,E2 -1481.157} C_VEL
LIN {X 0,Y 587.332,Z 322.325,A -85,B 0,C 180,E1 -1484.113,E2 -1484.113} C_VEL
LIN {X 0,Y 587.326,Z 322.322,A -85,B 0,C 180,E1 -1486.994,E2 -1486.994} C_VEL
LIN {X 0,Y 587.314,Z 322.331,A -85,B 0,C 180,E1 -1489.745,E2 -1489.745} C_VEL
LIN {X 0,Y 587.348,Z 322.321,A -85,B 0,C 180,E1 -1492.392,E2 -1492.392} C_VEL
LIN {X 0,Y 587.339,Z 322.403,A -85,B 0,C 180,E1 -1493.625,E2 -1493.625} C_VEL
LIN {X 0,Y 587.948,Z 325.829,A -85,B 0,C 180,E1 -1494.374,E2 -1494.374} C_VEL
LIN {X 0,Y 587.852,Z 337.797,A -85,B 0,C 180,E1 -1496.812,E2 -1496.812} C_VEL
LIN {X 0,Y 587.821,Z 351.045,A -85,B 0,C 180,E1 -1499.411,E2 -1499.411} C_VEL
LIN {X 0,Y 587.855,Z 365.903,A -85,B 0,C 180,E1 -1502.214,E2 -1502.214} C_VEL
LIN {X 0,Y 587.715,Z 379.58,A -85,B 0,C 180,E1 -1504.88,E2 -1504.88} C_VEL
LIN {X 0,Y 587.614,Z 393.275,A -85,B 0,C 180,E1 -1507.497,E2 -1507.497} C_VEL
LIN {X 0,Y 587.521,Z 408.926,A -85,B 0,C 180,E1 -1510.431,E2 -1510.431} C_VEL
LIN {X 0,Y 587.429,Z 424.578,A -85,B 0,C 180,E1 -1513.313,E2 -1513.313} C_VEL
LIN {X 0,Y 587.353,Z 440.229,A -85,B 0,C 180,E1 -1516.154,E2 -1516.154} C_VEL
LIN {X 0,Y 587.317,Z 449.156,A -85,B 0,C 180,E1 -1517.759,E2 -1517.759} C_VEL
LIN {X 0,Y 587.745,Z 454.938,A -85,B 0,C 180,E1 -1517.855,E2 -1517.855} C_VEL
LIN {X 0,Y 587.672,Z 468.213,A -85,B 0,C 180,E1 -1518.16,E2 -1518.16} C_VEL
LIN {X 0,Y 587.624,Z 480.635,A -85,B 0,C 180,E1 -1518.585,E2 -1518.585} C_VEL
LIN {X 0,Y 587.556,Z 492.629,A -85,B 0,C 180,E1 -1519.141,E2 -1519.141} C_VEL
LIN {X 0,Y 587.466,Z 504.199,A -85,B 0,C 180,E1 -1519.836,E2 -1519.836} C_VEL
LIN {X 0,Y 587.367,Z 514.596,A -85,B 0,C 180,E1 -1520.617,E2 -1520.617} C_VEL
LIN {X 0,Y 587.322,Z 523.111,A -85,B 0,C 180,E1 -1521.397,E2 -1521.397} C_VEL
LIN {X 0,Y 587.274,Z 530.959,A -85,B 0,C 180,E1 -1522.263,E2 -1522.263} C_VEL
LIN {X 0,Y 587.23,Z 537.469,A -85,B 0,C 180,E1 -1523.126,E2 -1523.126} C_VEL
LIN {X 0,Y 587.236,Z 543.866,A -85,B 0,C 180,E1 -1524.161,E2 -1524.161} C_VEL
LIN {X 0,Y 587.147,Z 548.95,A -85,B 0,C 180,E1 -1525.194,E2 -1525.194} C_VEL
LIN {X 0,Y 587.212,Z 552.895,A -85,B 0,C 180,E1 -1526.226,E2 -1526.226} C_VEL
LIN {X 0,Y 587.132,Z 555.808,A -85,B 0,C 180,E1 -1527.256,E2 -1527.256} C_VEL
LIN {X 0,Y 587.141,Z 557.2,A -85,B 0,C 180,E1 -1527.942,E2 -1527.942} C_VEL
LIN {X 0,Y 587.14,Z 558.784,A -85,B 0,C 180,E1 -1529.314,E2 -1529.314} C_VEL
LIN {X 0,Y 587.137,Z 559,A -85,B 0,C 180,E1 -1530,E2 -1530} C_VEL
LIN {X 0,Y 587.147,Z 558.185,A -85,B 0,C 180,E1 -1531.372,E2 -1531.372} C_VEL
LIN {X 0,Y 587.141,Z 557.201,A -85,B 0,C 180,E1 -1532.058,E2 -1532.058} C_VEL
LIN {X 0,Y 587.132,Z 555.81,A -85,B 0,C 180,E1 -1532.744,E2 -1532.744} C_VEL
LIN {X 0,Y 587.212,Z 552.896,A -85,B 0,C 180,E1 -1533.774,E2 -1533.774} C_VEL
LIN {X 0,Y 587.147,Z 548.95,A -85,B 0,C 180,E1 -1534.806,E2 -1534.806} C_VEL
LIN {X 0,Y 587.217,Z 542.877,A -85,B 0,C 180,E1 -1536.011,E2 -1536.011} C_VEL
LIN {X 0,Y 587.245,Z 536.236,A -85,B 0,C 180,E1 -1537.046,E2 -1537.046} C_VEL
LIN {X 0,Y 587.299,Z 527.99,A -85,B 0,C 180,E1 -1538.083,E2 -1538.083} C_VEL
LIN {X 0,Y 587.343,Z 519.537,A -85,B 0,C 180,E1 -1538.949,E2 -1538.949} C_VEL
LIN {X 0,Y 587.422,Z 509.094,A -85,B 0,C 180,E1 -1539.816,E2 -1539.816} C_VEL
LIN {X 0,Y 587.486,Z 498.758,A -85,B 0,C 180,E1 -1540.512,E2 -1540.512} C_VEL
LIN {X 0,Y 587.561,Z 486.818,A -85,B 0,C 180,E1 -1541.149,E2 -1541.149} C_VEL
LIN {X 0,Y 587.632,Z 474.599,A -85,B 0,C 180,E1 -1541.639,E2 -1541.639} C_VEL
LIN {X 0,Y 587.713,Z 461.434,A -85,B 0,C 180,E1 -1542.014,E2 -1542.014} C_VEL
LIN {X 0,Y 587.522,Z 450.597,A -85,B 0,C 180,E1 -1542.215,E2 -1542.215} C_VEL
LIN {X 0,Y 587.322,Z 449.034,A -85,B 0,C 180,E1 -1542.263,E2 -1542.263} C_VEL
LIN {X 0,Y 587.359,Z 434.361,A -85,B 0,C 180,E1 -1544.907,E2 -1544.907} C_VEL
LIN {X 0,Y 587.454,Z 418.709,A -85,B 0,C 180,E1 -1547.762,E2 -1547.762} C_VEL
LIN {X 0,Y 587.559,Z 403.058,A -85,B 0,C 180,E1 -1550.662,E2 -1550.662} C_VEL
LIN {X 0,Y 587.651,Z 389.363,A -85,B 0,C 180,E1 -1553.245,E2 -1553.245} C_VEL
LIN {X 0,Y 587.772,Z 375.668,A -85,B 0,C 180,E1 -1555.877,E2 -1555.877} C_VEL
LIN {X 0,Y 587.84,Z 363.762,A -85,B 0,C 180,E1 -1558.18,E2 -1558.18} C_VEL
LIN {X 0,Y 587.63,Z 347.921,A -85,B 0,C 180,E1 -1560.949,E2 -1560.949} C_VEL
LIN {X 0,Y 587.524,Z 329.812,A -85,B 0,C 180,E1 -1564.209,E2 -1564.209} C_VEL
LIN {X 0,Y 587.433,Z 322.672,A -85,B 0,C 180,E1 -1565.556,E2 -1565.556} C_VEL
LIN {X 0,Y 587.358,Z 322.325,A -85,B 0,C 180,E1 -1565.691,E2 -1565.691} C_VEL
LIN {X 0,Y 587.333,Z 322.326,A -85,B 0,C 180,E1 -1568.479,E2 -1568.479} C_VEL
LIN {X 0,Y 587.34,Z 322.324,A -85,B 0,C 180,E1 -1571.157,E2 -1571.157} C_VEL
LIN {X 0,Y 587.331,Z 322.326,A -85,B 0,C 180,E1 -1574.113,E2 -1574.113} C_VEL
LIN {X 0,Y 587.316,Z 322.328,A -85,B 0,C 180,E1 -1576.993,E2 -1576.993} C_VEL
LIN {X 0,Y 587.316,Z 322.327,A -85,B 0,C 180,E1 -1579.746,E2 -1579.746} C_VEL
LIN {X 0,Y 587.35,Z 322.322,A -85,B 0,C 180,E1 -1582.392,E2 -1582.392} C_VEL
LIN {X 0,Y 587.36,Z 322.325,A -85,B 0,C 180,E1 -1585.651,E2 -1585.651} C_VEL
LIN {X 0,Y 587.355,Z 322.323,A -85,B 0,C 180,E1 -1588.232,E2 -1588.232} C_VEL
LIN {X 0,Y 587.355,Z 322.321,A -85,B 0,C 180,E1 -1590.867,E2 -1590.867} C_VEL
LIN {X 0,Y 587.342,Z 322.323,A -85,B 0,C 180,E1 -1593.721,E2 -1593.721} C_VEL
LIN {X 0,Y 587.334,Z 322.324,A -85,B 0,C 180,E1 -1595.993,E2 -1595.993} C_VEL
LIN {X 0,Y 587.326,Z 322.328,A -85,B 0,C 180,E1 -1598.226,E2 -1598.226} C_VEL
LIN {X 0,Y 587.355,Z 322.326,A -85,B 0,C 180,E1 -1601.151,E2 -1601.151} C_VEL
LIN {X 0,Y 587.327,Z 322.33,A -85,B 0,C 180,E1 -1604.025,E2 -1604.025} C_VEL
LIN {X 0,Y 587.364,Z 322.32,A -85,B 0,C 180,E1 -1606.154,E2 -1606.154} C_VEL
LIN {X 0,Y 587.361,Z 322.321,A -85,B 0,C 180,E1 -1607.321,E2 -1607.321} C_VEL
LIN {X 0,Y 587.642,Z 326.744,A -85,B 0,C 180,E1 -1607.481,E2 -1607.481} C_VEL
LIN {X 0,Y 587.578,Z 339.05,A -85,B 0,C 180,E1 -1608.005,E2 -1608.005} C_VEL
LIN {X 0,Y 587.474,Z 350.098,A -85,B 0,C 180,E1 -1608.616,E2 -1608.616} C_VEL
LIN {X 0,Y 587.417,Z 361.37,A -85,B 0,C 180,E1 -1609.4,E2 -1609.4} C_VEL
LIN {X 0,Y 587.358,Z 370.442,A -85,B 0,C 180,E1 -1610.183,E2 -1610.183} C_VEL
LIN {X 0,Y 587.288,Z 380.246,A -85,B 0,C 180,E1 -1611.224,E2 -1611.224} C_VEL
LIN {X 0,Y 587.24,Z 388.083,A -85,B 0,C 180,E1 -1612.262,E2 -1612.262} C_VEL
LIN {X 0,Y 587.203,Z 394.971,A -85,B 0,C 180,E1 -1613.414,E2 -1613.414} C_VEL
LIN {X 0,Y 587.2,Z 400.058,A -85,B 0,C 180,E1 -1614.505,E2 -1614.505} C_VEL
LIN {X 0,Y 587.189,Z 403.728,A -85,B 0,C 180,E1 -1615.538,E2 -1615.538} C_VEL
LIN {X 0,Y 587.183,Z 406.388,A -85,B 0,C 180,E1 -1616.569,E2 -1616.569} C_VEL
LIN {X 0,Y 587.137,Z 408.486,A -85,B 0,C 180,E1 -1617.942,E2 -1617.942} C_VEL
LIN {X 0,Y 587.149,Z 408.912,A -85,B 0,C 180,E1 -1618.628,E2 -1618.628} C_VEL
LIN {X 0,Y 587.138,Z 408.602,A -85,B 0,C 180,E1 -1620,E2 -1620} C_VEL
LIN {X 0,Y 587.141,Z 407.865,A -85,B 0,C 180,E1 -1620.686,E2 -1620.686} C_VEL
LIN {X 0,Y 587.149,Z 406.698,A -85,B 0,C 180,E1 -1621.372,E2 -1621.372} C_VEL
LIN {X 0,Y 587.147,Z 405.124,A -85,B 0,C 180,E1 -1622.058,E2 -1622.058} C_VEL
LIN {X 0,Y 587.183,Z 401.956,A -85,B 0,C 180,E1 -1623.087,E2 -1623.087} C_VEL
LIN {X 0,Y 587.183,Z 397.736,A -85,B 0,C 180,E1 -1624.118,E2 -1624.118} C_VEL
LIN {X 0,Y 587.198,Z 391.322,A -85,B 0,C 180,E1 -1625.322,E2 -1625.322} C_VEL
LIN {X 0,Y 587.268,Z 383.867,A -85,B 0,C 180,E1 -1626.415,E2 -1626.415} C_VEL
LIN {X 0,Y 587.299,Z 375.576,A -85,B 0,C 180,E1 -1627.391,E2 -1627.391} C_VEL
LIN {X 0,Y 587.404,Z 365.635,A -85,B 0,C 180,E1 -1628.341,E2 -1628.341} C_VEL
LIN {X 0,Y 587.457,Z 355.489,A -85,B 0,C 180,E1 -1629.121,E2 -1629.121} C_VEL
LIN {X 0,Y 587.531,Z 344.268,A -85,B 0,C 180,E1 -1629.814,E2 -1629.814} C_VEL
LIN {X 0,Y 587.617,Z 332.639,A -85,B 0,C 180,E1 -1630.378,E2 -1630.378} C_VEL
LIN {X 0,Y 587.415,Z 322.737,A -85,B 0,C 180,E1 -1630.752,E2 -1630.752} C_VEL
LIN {X 0,Y 587.353,Z 322.32,A -85,B 0,C 180,E1 -1630.775,E2 -1630.775} C_VEL
LIN {X 0,Y 587.367,Z 322.324,A -85,B 0,C 180,E1 -1633.845,E2 -1633.845} C_VEL
LIN {X 0,Y 587.322,Z 322.324,A -85,B 0,C 180,E1 -1635.819,E2 -1635.819} C_VEL
LIN {X 0,Y 586.665,Z 322.408,A -85,B 0,C 180,E1 -1636.392,E2 -1636.392} C_VEL
LIN {X 0,Y 583.787,Z 322.771,A -85,B 0,C 180,E1 -1637.32,E2 -1637.32} C_VEL
LIN {X 0,Y 581.364,Z 323.067,A -85,B 0,C 180,E1 -1638.067,E2 -1638.067} C_VEL
LIN {X 0,Y 580.347,Z 323.193,A -85,B 0,C 180,E1 -1638.644,E2 -1638.644} C_VEL
LIN {X 0,Y 580.277,Z 323.204,A -85,B 0,C 180,E1 -1638.84,E2 -1638.84} C_VEL
LIN {X 0,Y 580.29,Z 323.2,A -85,B 0,C 180,E1 -1641.305,E2 -1641.305} C_VEL
LIN {X 0,Y 580.303,Z 323.204,A -85,B 0,C 180,E1 -1644.316,E2 -1644.316} C_VEL
LIN {X 0,Y 580.28,Z 323.202,A -85,B 0,C 180,E1 -1646.623,E2 -1646.623} C_VEL
LIN {X 0,Y 580.306,Z 323.199,A -85,B 0,C 180,E1 -1649.31,E2 -1649.31} C_VEL
LIN {X 0,Y 580.305,Z 323.196,A -85,B 0,C 180,E1 -1652.2,E2 -1652.2} C_VEL
LIN {X 0,Y 580.294,Z 323.201,A -85,B 0,C 180,E1 -1654.696,E2 -1654.696} C_VEL
LIN {X 0,Y 580.302,Z 323.198,A -85,B 0,C 180,E1 -1657.268,E2 -1657.268} C_VEL
LIN {X 0,Y 580.302,Z 323.204,A -85,B 0,C 180,E1 -1660.271,E2 -1660.271} C_VEL
LIN {X 0,Y 580.28,Z 323.2,A -85,B 0,C 180,E1 -1662.706,E2 -1662.706} C_VEL
LIN {X 0,Y 580.277,Z 323.207,A -85,B 0,C 180,E1 -1665.608,E2 -1665.608} C_VEL
LIN {X 0,Y 580.317,Z 323.195,A -85,B 0,C 180,E1 -1668.234,E2 -1668.234} C_VEL
LIN {X 0,Y 580.282,Z 323.207,A -85,B 0,C 180,E1 -1670.965,E2 -1670.965} C_VEL
LIN {X 0,Y 580.269,Z 323.2,A -85,B 0,C 180,E1 -1673.596,E2 -1673.596} C_VEL
LIN {X 0,Y 580.32,Z 323.201,A -85,B 0,C 180,E1 -1676.145,E2 -1676.145} C_VEL
LIN {X 0,Y 580.28,Z 323.2,A -85,B 0,C 180,E1 -1678.615,E2 -1678.615} C_VEL
LIN {X 0,Y 580.296,Z 323.199,A -85,B 0,C 180,E1 -1681.024,E2 -1681.024} C_VEL
LIN {X 0,Y 580.294,Z 323.201,A -85,B 0,C 180,E1 -1683.666,E2 -1683.666} C_VEL
LIN {X 0,Y 580.302,Z 323.198,A -85,B 0,C 180,E1 -1685.684,E2 -1685.684} C_VEL
LIN {X 0,Y 580.276,Z 323.2,A -85,B 0,C 180,E1 -1687.947,E2 -1687.947} C_VEL
LIN {X 0,Y 580.302,Z 323.198,A -85,B 0,C 180,E1 -1690.913,E2 -1690.913} C_VEL
LIN {X 0,Y 580.283,Z 323.205,A -85,B 0,C 180,E1 -1693.826,E2 -1693.826} C_VEL
LIN {X 0,Y 580.328,Z 323.198,A -85,B 0,C 180,E1 -1695.983,E2 -1695.983} C_VEL
LIN {X 0,Y 580.307,Z 323.198,A -85,B 0,C 180,E1 -1698.827,E2 -1698.827} C_VEL
LIN {X 0,Y 580.329,Z 323.194,A -85,B 0,C 180,E1 -1701.644,E2 -1701.644} C_VEL
LIN {X 0,Y 580.336,Z 323.198,A -85,B 0,C 180,E1 -1704.44,E2 -1704.44} C_VEL
LIN {X 0,Y 580.345,Z 323.196,A -85,B 0,C 180,E1 -1707.918,E2 -1707.918} C_VEL
LIN {X 0,Y 580.361,Z 323.189,A -85,B 0,C 180,E1 -1710.694,E2 -1710.694} C_VEL
LIN {X 0,Y 580.292,Z 323.206,A -85,B 0,C 180,E1 -1713.472,E2 -1713.472} C_VEL
LIN {X 0,Y 580.336,Z 323.195,A -85,B 0,C 180,E1 -1715.56,E2 -1715.56} C_VEL
LIN {X 0,Y 580.335,Z 323.195,A -85,B 0,C 180,E1 -1718.356,E2 -1718.356} C_VEL
LIN {X 0,Y 580.302,Z 323.197,A -85,B 0,C 180,E1 -1721.191,E2 -1721.191} C_VEL
LIN {X 0,Y 580.328,Z 323.201,A -85,B 0,C 180,E1 -1724.017,E2 -1724.017} C_VEL
LIN {X 0,Y 580.314,Z 323.195,A -85,B 0,C 180,E1 -1726.914,E2 -1726.914} C_VEL
LIN {X 0,Y 580.307,Z 323.198,A -85,B 0,C 180,E1 -1729.822,E2 -1729.822} C_VEL
LIN {X 0,Y 580.298,Z 323.204,A -85,B 0,C 180,E1 -1732.803,E2 -1732.803} C_VEL
LIN {X 0,Y 580.31,Z 323.198,A -85,B 0,C 180,E1 -1735.08,E2 -1735.08} C_VEL
LIN {X 0,Y 580.303,Z 323.204,A -85,B 0,C 180,E1 -1738.186,E2 -1738.186} C_VEL
LIN {X 0,Y 580.286,Z 323.199,A -85,B 0,C 180,E1 -1740.695,E2 -1740.695} C_VEL
LIN {X 0,Y 580.307,Z 323.201,A -85,B 0,C 180,E1 -1743.317,E2 -1743.317} C_VEL
LIN {X 0,Y 580.248,Z 323.205,A -85,B 0,C 180,E1 -1745.757,E2 -1745.757} C_VEL
LIN {X 0,Y 580.291,Z 323.198,A -85,B 0,C 180,E1 -1748.147,E2 -1748.147} C_VEL
LIN {X 0,Y 580.301,Z 323.201,A -85,B 0,C 180,E1 -1750.844,E2 -1750.844} C_VEL
LIN {X 0,Y 580.292,Z 323.2,A -85,B 0,C 180,E1 -1753.657,E2 -1753.657} C_VEL
LIN {X 0,Y 580.281,Z 323.2,A -85,B 0,C 180,E1 -1756.61,E2 -1756.61} C_VEL
LIN {X 0,Y 580.301,Z 323.2,A -85,B 0,C 180,E1 -1759.157,E2 -1759.157} C_VEL
LIN {X 0,Y 580.293,Z 323.198,A -85,B 0,C 180,E1 -1761.927,E2 -1761.927} C_VEL
LIN {X 0,Y 580.26,Z 323.205,A -85,B 0,C 180,E1 -1764.453,E2 -1764.453} C_VEL
LIN {X 0,Y 580.294,Z 323.2,A -85,B 0,C 180,E1 -1766.975,E2 -1766.975} C_VEL
LIN {X 0,Y 580.3,Z 323.198,A -85,B 0,C 180,E1 -1769.425,E2 -1769.425} C_VEL
LIN {X 0,Y 580.302,Z 323.2,A -85,B 0,C 180,E1 -1772.142,E2 -1772.142} C_VEL
LIN {X 0,Y 580.327,Z 323.2,A -85,B 0,C 180,E1 -1775.27,E2 -1775.27} C_VEL
LIN {X 0,Y 580.274,Z 323.2,A -85,B 0,C 180,E1 -1777.948,E2 -1777.948} C_VEL
LIN {X 0,Y 580.301,Z 323.201,A -85,B 0,C 180,E1 -1780.914,E2 -1780.914} C_VEL
LIN {X 0,Y 580.277,Z 323.202,A -85,B 0,C 180,E1 -1783.826,E2 -1783.826} C_VEL
LIN {X 0,Y 580.333,Z 323.2,A -85,B 0,C 180,E1 -1785.983,E2 -1785.983} C_VEL
LIN {X 0,Y 580.312,Z 323.196,A -85,B 0,C 180,E1 -1788.827,E2 -1788.827} C_VEL
LIN {X 0,Y 580.338,Z 323.195,A -85,B 0,C 180,E1 -1791.644,E2 -1791.644} C_VEL
LIN {X 0,Y 580.328,Z 323.196,A -85,B 0,C 180,E1 -1794.44,E2 -1794.44} C_VEL
LIN {X 0,Y 580.343,Z 323.192,A -85,B 0,C 180,E1 -1797.224,E2 -1797.224} C_VEL
LIN {X 0,Y 580.359,Z 323.195,A -85,B 0,C 180,E1 -1800,E2 -1800} C_VEL
LIN {X 0,Y 580.344,Z 323.191,A -85,B 0,C 180,E1 -1802.777,E2 -1802.777} C_VEL
LIN {X 0,Y 580.324,Z 323.201,A -85,B 0,C 180,E1 -1805.56,E2 -1805.56} C_VEL
LIN {X 0,Y 580.329,Z 323.196,A -85,B 0,C 180,E1 -1807.655,E2 -1807.655} C_VEL
LIN {X 0,Y 580.306,Z 323.2,A -85,B 0,C 180,E1 -1810.467,E2 -1810.467} C_VEL
LIN {X 0,Y 580.277,Z 323.2,A -85,B 0,C 180,E1 -1813.304,E2 -1813.304} C_VEL
LIN {X 0,Y 580.298,Z 323.197,A -85,B 0,C 180,E1 -1815.453,E2 -1815.453} C_VEL
LIN {X 0,Y 580.306,Z 323.201,A -85,B 0,C 180,E1 -1817.624,E2 -1817.624} C_VEL
LIN {X 0,Y 580.309,Z 323.201,A -85,B 0,C 180,E1 -1819.822,E2 -1819.822} C_VEL
LIN {X 0,Y 580.296,Z 323.2,A -85,B 0,C 180,E1 -1822.803,E2 -1822.803} C_VEL
LIN {X 0,Y 580.31,Z 323.202,A -85,B 0,C 180,E1 -1825.08,E2 -1825.08} C_VEL
LIN {X 0,Y 580.306,Z 323.2,A -85,B 0,C 180,E1 -1828.185,E2 -1828.185} C_VEL
LIN {X 0,Y 580.29,Z 323.2,A -85,B 0,C 180,E1 -1830.694,E2 -1830.694} C_VEL
LIN {X 0,Y 580.307,Z 323.197,A -85,B 0,C 180,E1 -1833.316,E2 -1833.316} C_VEL
LIN {X 0,Y 580.265,Z 323.206,A -85,B 0,C 180,E1 -1835.758,E2 -1835.758} C_VEL
LIN {X 0,Y 580.294,Z 323.198,A -85,B 0,C 180,E1 -1838.146,E2 -1838.146} C_VEL
LIN {X 0,Y 580.303,Z 323.204,A -85,B 0,C 180,E1 -1840.843,E2 -1840.843} C_VEL
LIN {X 0,Y 580.283,Z 323.199,A -85,B 0,C 180,E1 -1843.658,E2 -1843.658} C_VEL
LIN {X 0,Y 580.291,Z 323.2,A -85,B 0,C 180,E1 -1846.608,E2 -1846.608} C_VEL
LIN {X 0,Y 580.301,Z 323.198,A -85,B 0,C 180,E1 -1849.156,E2 -1849.156} C_VEL
LIN {X 0,Y 580.293,Z 323.203,A -85,B 0,C 180,E1 -1851.927,E2 -1851.927} C_VEL
LIN {X 0,Y 580.309,Z 323.301,A -85,B 0,C 180,E1 -1853.385,E2 -1853.385} C_VEL
LIN {X 0,Y 581.111,Z 328.432,A -85,B 0,C 180,E1 -1854.513,E2 -1854.513} C_VEL
LIN {X 0,Y 580.9,Z 342.534,A -85,B 0,C 180,E1 -1857.426,E2 -1857.426} C_VEL
LIN {X 0,Y 580.878,Z 357.053,A -85,B 0,C 180,E1 -1860.26,E2 -1860.26} C_VEL
LIN {X 0,Y 580.888,Z 371.595,A -85,B 0,C 180,E1 -1863.018,E2 -1863.018} C_VEL
LIN {X 0,Y 580.749,Z 385.449,A -85,B 0,C 180,E1 -1865.704,E2 -1865.704} C_VEL
LIN {X 0,Y 580.609,Z 399.144,A -85,B 0,C 180,E1 -1868.334,E2 -1868.334} C_VEL
LIN {X 0,Y 580.484,Z 414.796,A -85,B 0,C 180,E1 -1871.286,E2 -1871.286} C_VEL
LIN {X 0,Y 580.355,Z 430.447,A -85,B 0,C 180,E1 -1874.188,E2 -1874.188} C_VEL
LIN {X 0,Y 580.242,Z 446.099,A -85,B 0,C 180,E1 -1877.051,E2 -1877.051} C_VEL
LIN {X 0,Y 580.273,Z 449.156,A -85,B 0,C 180,E1 -1877.608,E2 -1877.608} C_VEL
LIN {X 0,Y 580.827,Z 454.938,A -85,B 0,C 180,E1 -1877.708,E2 -1877.708} C_VEL
LIN {X 0,Y 580.746,Z 468.214,A -85,B 0,C 180,E1 -1878.017,E2 -1878.017} C_VEL
LIN {X 0,Y 580.665,Z 480.368,A -85,B 0,C 180,E1 -1878.436,E2 -1878.436} C_VEL
LIN {X 0,Y 580.579,Z 492.628,A -85,B 0,C 180,E1 -1879.009,E2 -1879.009} C_VEL
LIN {X 0,Y 580.443,Z 504.2,A -85,B 0,C 180,E1 -1879.712,E2 -1879.712} C_VEL
LIN {X 0,Y 580.347,Z 514.597,A -85,B 0,C 180,E1 -1880.503,E2 -1880.503} C_VEL
LIN {X 0,Y 580.271,Z 523.111,A -85,B 0,C 180,E1 -1881.292,E2 -1881.292} C_VEL
LIN {X 0,Y 580.222,Z 530.96,A -85,B 0,C 180,E1 -1882.168,E2 -1882.168} C_VEL
LIN {X 0,Y 580.154,Z 538.65,A -85,B 0,C 180,E1 -1883.222,E2 -1883.222} C_VEL
LIN {X 0,Y 580.139,Z 545.68,A -85,B 0,C 180,E1 -1884.438,E2 -1884.438} C_VEL
LIN {X 0,Y 580.108,Z 550.371,A -85,B 0,C 180,E1 -1885.483,E2 -1885.483} C_VEL
LIN {X 0,Y 580.123,Z 553.957,A -85,B 0,C 180,E1 -1886.527,E2 -1886.527} C_VEL
LIN {X 0,Y 580.043,Z 555.808,A -85,B 0,C 180,E1 -1887.222,E2 -1887.222} C_VEL
LIN {X 0,Y 580.04,Z 557.2,A -85,B 0,C 180,E1 -1887.917,E2 -1887.917} C_VEL
LIN {X 0,Y 580.04,Z 558.784,A -85,B 0,C 180,E1 -1889.306,E2 -1889.306} C_VEL
LIN {X 0,Y 580.037,Z 559,A -85,B 0,C 180,E1 -1890,E2 -1890} C_VEL
LIN {X 0,Y 580.047,Z 558.186,A -85,B 0,C 180,E1 -1891.389,E2 -1891.389} C_VEL
LIN {X 0,Y 580.04,Z 557.201,A -85,B 0,C 180,E1 -1892.083,E2 -1892.083} C_VEL
LIN {X 0,Y 580.043,Z 555.81,A -85,B 0,C 180,E1 -1892.778,E2 -1892.778} C_VEL
LIN {X 0,Y 580.109,Z 552.896,A -85,B 0,C 180,E1 -1893.821,E2 -1893.821} C_VEL
LIN {X 0,Y 580.054,Z 548.949,A -85,B 0,C 180,E1 -1894.865,E2 -1894.865} C_VEL
LIN {X 0,Y 580.139,Z 542.877,A -85,B 0,C 180,E1 -1896.085,E2 -1896.085} C_VEL
LIN {X 0,Y 580.184,Z 536.237,A -85,B 0,C 180,E1 -1897.132,E2 -1897.132} C_VEL
LIN {X 0,Y 580.25,Z 527.99,A -85,B 0,C 180,E1 -1898.182,E2 -1898.182} C_VEL
LIN {X 0,Y 580.308,Z 519.537,A -85,B 0,C 180,E1 -1899.058,E2 -1899.058} C_VEL
LIN {X 0,Y 580.425,Z 509.095,A -85,B 0,C 180,E1 -1899.936,E2 -1899.936} C_VEL
LIN {X 0,Y 580.491,Z 498.756,A -85,B 0,C 180,E1 -1900.64,E2 -1900.64} C_VEL
LIN {X 0,Y 580.596,Z 487.249,A -85,B 0,C 180,E1 -1901.264,E2 -1901.264} C_VEL
LIN {X 0,Y 580.692,Z 474.47,A -85,B 0,C 180,E1 -1901.785,E2 -1901.785} C_VEL
LIN {X 0,Y 580.786,Z 461.433,A -85,B 0,C 180,E1 -1902.159,E2 -1902.159} C_VEL
LIN {X 0,Y 580.634,Z 451.539,A -85,B 0,C 180,E1 -1902.348,E2 -1902.348} C_VEL
LIN {X 0,Y 580.256,Z 449.034,A -85,B 0,C 180,E1 -1902.415,E2 -1902.415} C_VEL
LIN {X 0,Y 580.342,Z 434.361,A -85,B 0,C 180,E1 -1905.092,E2 -1905.092} C_VEL
LIN {X 0,Y 580.437,Z 418.709,A -85,B 0,C 180,E1 -1907.984,E2 -1907.984} C_VEL
LIN {X 0,Y 580.588,Z 403.2,A -85,B 0,C 180,E1 -1910.895,E2 -1910.895} C_VEL
LIN {X 0,Y 580.732,Z 387.406,A -85,B 0,C 180,E1 -1913.917,E2 -1913.917} C_VEL
LIN {X 0,Y 580.869,Z 372.608,A -85,B 0,C 180,E1 -1916.788,E2 -1916.788} C_VEL
LIN {X 0,Y 580.707,Z 356.981,A -85,B 0,C 180,E1 -1919.533,E2 -1919.533} C_VEL
LIN {X 0,Y 580.49,Z 342.14,A -85,B 0,C 180,E1 -1922.189,E2 -1922.189} C_VEL
LIN {X 0,Y 580.603,Z 326.526,A -85,B 0,C 180,E1 -1925.098,E2 -1925.098} C_VEL
LIN {X 0,Y 580.335,Z 323.2,A -85,B 0,C 180,E1 -1925.768,E2 -1925.768} C_VEL
LIN {X 0,Y 580.292,Z 323.202,A -85,B 0,C 180,E1 -1928.146,E2 -1928.146} C_VEL
LIN {X 0,Y 580.301,Z 323.2,A -85,B 0,C 180,E1 -1930.844,E2 -1930.844} C_VEL
LIN {X 0,Y 580.284,Z 323.202,A -85,B 0,C 180,E1 -1933.658,E2 -1933.658} C_VEL
LIN {X 0,Y 580.28,Z 323.202,A -85,B 0,C 180,E1 -1936.609,E2 -1936.609} C_VEL
LIN {X 0,Y 580.303,Z 323.2,A -85,B 0,C 180,E1 -1939.157,E2 -1939.157} C_VEL
LIN {X 0,Y 580.295,Z 323.201,A -85,B 0,C 180,E1 -1941.927,E2 -1941.927} C_VEL
LIN {X 0,Y 580.287,Z 323.205,A -85,B 0,C 180,E1 -1944.455,E2 -1944.455} C_VEL
LIN {X 0,Y 580.294,Z 323.204,A -85,B 0,C 180,E1 -1946.975,E2 -1946.975} C_VEL
LIN {X 0,Y 580.308,Z 323.199,A -85,B 0,C 180,E1 -1949.426,E2 -1949.426} C_VEL
LIN {X 0,Y 580.303,Z 323.199,A -85,B 0,C 180,E1 -1952.141,E2 -1952.141} C_VEL
LIN {X 0,Y 580.327,Z 323.198,A -85,B 0,C 180,E1 -1955.27,E2 -1955.27} C_VEL
LIN {X 0,Y 580.276,Z 323.204,A -85,B 0,C 180,E1 -1957.947,E2 -1957.947} C_VEL
LIN {X 0,Y 580.304,Z 323.202,A -85,B 0,C 180,E1 -1960.913,E2 -1960.913} C_VEL
LIN {X 0,Y 580.277,Z 323.206,A -85,B 0,C 180,E1 -1963.825,E2 -1963.825} C_VEL
LIN {X 0,Y 580.331,Z 323.197,A -85,B 0,C 180,E1 -1965.983,E2 -1965.983} C_VEL
LIN {X 0,Y 580.315,Z 323.221,A -85,B 0,C 180,E1 -1967.209,E2 -1967.209} C_VEL
LIN {X 0,Y 580.678,Z 326.406,A -85,B 0,C 180,E1 -1967.328,E2 -1967.328} C_VEL
LIN {X 0,Y 580.605,Z 338.818,A -85,B 0,C 180,E1 -1967.859,E2 -1967.859} C_VEL
LIN {X 0,Y 580.463,Z 350.927,A -85,B 0,C 180,E1 -1968.54,E2 -1968.54} C_VEL
LIN {X 0,Y 580.414,Z 361.334,A -85,B 0,C 180,E1 -1969.28,E2 -1969.28} C_VEL
LIN {X 0,Y 580.315,Z 370.319,A -85,B 0,C 180,E1 -1970.062,E2 -1970.062} C_VEL
LIN {X 0,Y 580.256,Z 378.654,A -85,B 0,C 180,E1 -1970.941,E2 -1970.941} C_VEL
LIN {X 0,Y 580.19,Z 386.808,A -85,B 0,C 180,E1 -1971.992,E2 -1971.992} C_VEL
LIN {X 0,Y 580.149,Z 393.353,A -85,B 0,C 180,E1 -1973.042,E2 -1973.042} C_VEL
LIN {X 0,Y 580.119,Z 398.55,A -85,B 0,C 180,E1 -1974.089,E2 -1974.089} C_VEL
LIN {X 0,Y 580.043,Z 402.59,A -85,B 0,C 180,E1 -1975.135,E2 -1975.135} C_VEL
LIN {X 0,Y 580.105,Z 404.709,A -85,B 0,C 180,E1 -1975.831,E2 -1975.831} C_VEL
LIN {X 0,Y 580.109,Z 406.365,A -85,B 0,C 180,E1 -1976.527,E2 -1976.527} C_VEL
LIN {X 0,Y 580.036,Z 408.474,A -85,B 0,C 180,E1 -1977.917,E2 -1977.917} C_VEL
LIN {X 0,Y 580.048,Z 408.91,A -85,B 0,C 180,E1 -1978.611,E2 -1978.611} C_VEL
LIN {X 0,Y 580.038,Z 408.61,A -85,B 0,C 180,E1 -1980,E2 -1980} C_VEL
LIN {X 0,Y 580.041,Z 407.881,A -85,B 0,C 180,E1 -1980.694,E2 -1980.694} C_VEL
LIN {X 0,Y 580.049,Z 406.721,A -85,B 0,C 180,E1 -1981.388,E2 -1981.388} C_VEL
LIN {X 0,Y 580.047,Z 405.156,A -85,B 0,C 180,E1 -1982.083,E2 -1982.083} C_VEL
LIN {X 0,Y 580.094,Z 402.001,A -85,B 0,C 180,E1 -1983.125,E2 -1983.125} C_VEL
LIN {X 0,Y 580.108,Z 397.793,A -85,B 0,C 180,E1 -1984.168,E2 -1984.168} C_VEL
LIN {X 0,Y 580.124,Z 391.391,A -85,B 0,C 180,E1 -1985.387,E2 -1985.387} C_VEL
LIN {X 0,Y 580.204,Z 384.489,A -85,B 0,C 180,E1 -1986.422,E2 -1986.422} C_VEL
LIN {X 0,Y 580.253,Z 375.687,A -85,B 0,C 180,E1 -1987.481,E2 -1987.481} C_VEL
LIN {X 0,Y 580.383,Z 365.77,A -85,B 0,C 180,E1 -1988.443,E2 -1988.443} C_VEL
LIN {X 0,Y 580.435,Z 355.661,A -85,B 0,C 180,E1 -1989.232,E2 -1989.232} C_VEL
LIN {X 0,Y 580.551,Z 344.481,A -85,B 0,C 180,E1 -1989.934,E2 -1989.934} C_VEL
LIN {X 0,Y 580.597,Z 333.898,A -85,B 0,C 180,E1 -1990.461,E2 -1990.461} C_VEL
LIN {X 0,Y 580.683,Z 325.818,A -85,B 0,C 180,E1 -1990.783,E2 -1990.783} C_VEL
LIN {X 0,Y 580.303,Z 323.198,A -85,B 0,C 180,E1 -1990.884,E2 -1990.884} C_VEL
LIN {X 0,Y 580.281,Z 323.202,A -85,B 0,C 180,E1 -1993.304,E2 -1993.304} C_VEL
LIN {X 0,Y 580.279,Z 323.202,A -85,B 0,C 180,E1 -1995.817,E2 -1995.817} C_VEL
LIN {X 0,Y 580.263,Z 323.201,A -85,B 0,C 180,E1 -1998.355,E2 -1998.355} C_VEL
LIN {X 0,Y 580.277,Z 323.204,A -85,B 0,C 180,E1 -1998.84,E2 -1998.84} C_VEL
LIN {X 0,Y 579.643,Z 323.287,A -85,B 0,C 180,E1 -1999.42,E2 -1999.42} C_VEL
LIN {X 0,Y 576.785,Z 323.641,A -85,B 0,C 180,E1 -2000.36,E2 -2000.36} C_VEL
LIN {X 0,Y 574.351,Z 323.942,A -85,B 0,C 180,E1 -2001.117,E2 -2001.117} C_VEL
LIN {X 0,Y 573.307,Z 324.068,A -85,B 0,C 180,E1 -2001.702,E2 -2001.702} C_VEL
LIN {X 0,Y 573.224,Z 324.079,A -85,B 0,C 180,E1 -2001.9,E2 -2001.9} C_VEL
LIN {X 0,Y 573.272,Z 324.074,A -85,B 0,C 180,E1 -2004.878,E2 -2004.878} C_VEL
LIN {X 0,Y 573.277,Z 324.077,A -85,B 0,C 180,E1 -2007.766,E2 -2007.766} C_VEL
LIN {X 0,Y 573.254,Z 324.077,A -85,B 0,C 180,E1 -2010.176,E2 -2010.176} C_VEL
LIN {X 0,Y 573.259,Z 324.075,A -85,B 0,C 180,E1 -2012.645,E2 -2012.645} C_VEL
LIN {X 0,Y 573.212,Z 324.085,A -85,B 0,C 180,E1 -2015.187,E2 -2015.187} C_VEL
LIN {X 0,Y 573.239,Z 324.076,A -85,B 0,C 180,E1 -2017.807,E2 -2017.807} C_VEL
LIN {X 0,Y 573.273,Z 324.077,A -85,B 0,C 180,E1 -2020.528,E2 -2020.528} C_VEL
LIN {X 0,Y 573.247,Z 324.081,A -85,B 0,C 180,E1 -2023.669,E2 -2023.669} C_VEL
LIN {X 0,Y 573.251,Z 324.075,A -85,B 0,C 180,E1 -2026.642,E2 -2026.642} C_VEL
LIN {X 0,Y 573.247,Z 324.079,A -85,B 0,C 180,E1 -2029.475,E2 -2029.475} C_VEL
LIN {X 0,Y 573.237,Z 324.078,A -85,B 0,C 180,E1 -2032.192,E2 -2032.192} C_VEL
LIN {X 0,Y 573.238,Z 324.077,A -85,B 0,C 180,E1 -2035.228,E2 -2035.228} C_VEL
LIN {X 0,Y 573.255,Z 324.079,A -85,B 0,C 180,E1 -2037.771,E2 -2037.771} C_VEL
LIN {X 0,Y 573.267,Z 324.073,A -85,B 0,C 180,E1 -2040.634,E2 -2040.634} C_VEL
LIN {X 0,Y 573.253,Z 324.078,A -85,B 0,C 180,E1 -2043.024,E2 -2043.024} C_VEL
LIN {X 0,Y 573.277,Z 324.076,A -85,B 0,C 180,E1 -2045.366,E2 -2045.366} C_VEL
LIN {X 0,Y 573.232,Z 324.082,A -85,B 0,C 180,E1 -2048.419,E2 -2048.419} C_VEL
LIN {X 0,Y 573.28,Z 324.074,A -85,B 0,C 180,E1 -2050.728,E2 -2050.728} C_VEL
LIN {X 0,Y 573.254,Z 324.078,A -85,B 0,C 180,E1 -2053.622,E2 -2053.622} C_VEL
LIN {X 0,Y 573.276,Z 324.079,A -85,B 0,C 180,E1 -2055.807,E2 -2055.807} C_VEL
LIN {X 0,Y 573.265,Z 324.075,A -85,B 0,C 180,E1 -2058.745,E2 -2058.745} C_VEL
LIN {X 0,Y 573.285,Z 324.072,A -85,B 0,C 180,E1 -2061.54,E2 -2061.54} C_VEL
LIN {X 0,Y 573.303,Z 324.074,A -85,B 0,C 180,E1 -2064.372,E2 -2064.372} C_VEL
LIN {X 0,Y 573.315,Z 324.071,A -85,B 0,C 180,E1 -2067.892,E2 -2067.892} C_VEL
LIN {X 0,Y 573.332,Z 324.065,A -85,B 0,C 180,E1 -2070.702,E2 -2070.702} C_VEL
LIN {X 0,Y 573.307,Z 324.069,A -85,B 0,C 180,E1 -2072.811,E2 -2072.811} C_VEL
LIN {X 0,Y 573.303,Z 324.071,A -85,B 0,C 180,E1 -2075.628,E2 -2075.628} C_VEL
LIN {X 0,Y 573.291,Z 324.074,A -85,B 0,C 180,E1 -2078.46,E2 -2078.46} C_VEL
LIN {X 0,Y 573.274,Z 324.072,A -85,B 0,C 180,E1 -2081.312,E2 -2081.312} C_VEL
LIN {X 0,Y 573.276,Z 324.078,A -85,B 0,C 180,E1 -2084.193,E2 -2084.193} C_VEL
LIN {X 0,Y 573.26,Z 324.075,A -85,B 0,C 180,E1 -2087.112,E2 -2087.112} C_VEL
LIN {X 0,Y 573.255,Z 324.075,A -85,B 0,C 180,E1 -2090.077,E2 -2090.077} C_VEL
LIN {X 0,Y 573.237,Z 324.082,A -85,B 0,C 180,E1 -2093.1,E2 -2093.1} C_VEL
LIN {X 0,Y 573.258,Z 324.075,A -85,B 0,C 180,E1 -2095.41,E2 -2095.41} C_VEL
LIN {X 0,Y 573.255,Z 324.08,A -85,B 0,C 180,E1 -2098.029,E2 -2098.029} C_VEL
LIN {X 0,Y 573.249,Z 324.08,A -85,B 0,C 180,E1 -2100.176,E2 -2100.176} C_VEL
LIN {X 0,Y 573.258,Z 324.074,A -85,B 0,C 180,E1 -2102.645,E2 -2102.645} C_VEL
LIN {X 0,Y 573.21,Z 324.086,A -85,B 0,C 180,E1 -2105.188,E2 -2105.188} C_VEL
LIN {X 0,Y 573.238,Z 324.077,A -85,B 0,C 180,E1 -2107.808,E2 -2107.808} C_VEL
LIN {X 0,Y 573.247,Z 324.082,A -85,B 0,C 180,E1 -2110.525,E2 -2110.525} C_VEL
LIN {X 0,Y 573.251,Z 324.075,A -85,B 0,C 180,E1 -2113.358,E2 -2113.358} C_VEL
LIN {X 0,Y 573.248,Z 324.078,A -85,B 0,C 180,E1 -2116.331,E2 -2116.331} C_VEL
LIN {X 0,Y 573.242,Z 324.076,A -85,B 0,C 180,E1 -2118.544,E2 -2118.544} C_VEL
LIN {X 0,Y 573.246,Z 324.082,A -85,B 0,C 180,E1 -2121.299,E2 -2121.299} C_VEL
LIN {X 0,Y 573.218,Z 324.079,A -85,B 0,C 180,E1 -2124.019,E2 -2124.019} C_VEL
LIN {X 0,Y 573.29,Z 324.077,A -85,B 0,C 180,E1 -2126.519,E2 -2126.519} C_VEL
LIN {X 0,Y 573.233,Z 324.077,A -85,B 0,C 180,E1 -2129.118,E2 -2129.118} C_VEL
LIN {X 0,Y 573.242,Z 324.079,A -85,B 0,C 180,E1 -2131.436,E2 -2131.436} C_VEL
LIN {X 0,Y 573.268,Z 324.078,A -85,B 0,C 180,E1 -2133.81,E2 -2133.81} C_VEL
LIN {X 0,Y 573.232,Z 324.077,A -85,B 0,C 180,E1 -2136.135,E2 -2136.135} C_VEL
LIN {X 0,Y 573.255,Z 324.078,A -85,B 0,C 180,E1 -2139.174,E2 -2139.174} C_VEL
LIN {X 0,Y 573.221,Z 324.079,A -85,B 0,C 180,E1 -2141.411,E2 -2141.411} C_VEL
LIN {X 0,Y 573.25,Z 324.076,A -85,B 0,C 180,E1 -2143.622,E2 -2143.622} C_VEL
LIN {X 0,Y 573.28,Z 324.077,A -85,B 0,C 180,E1 -2145.807,E2 -2145.807} C_VEL
LIN {X 0,Y 573.269,Z 324.073,A -85,B 0,C 180,E1 -2148.745,E2 -2148.745} C_VEL
LIN {X 0,Y 573.295,Z 324.074,A -85,B 0,C 180,E1 -2151.541,E2 -2151.541} C_VEL
LIN {X 0,Y 573.295,Z 324.071,A -85,B 0,C 180,E1 -2154.372,E2 -2154.372} C_VEL
LIN {X 0,Y 573.309,Z 324.069,A -85,B 0,C 180,E1 -2157.893,E2 -2157.893} C_VEL
LIN {X 0,Y 573.336,Z 324.066,A -85,B 0,C 180,E1 -2160.702,E2 -2160.702} C_VEL
LIN {X 0,Y 573.31,Z 324.068,A -85,B 0,C 180,E1 -2162.811,E2 -2162.811} C_VEL
LIN {X 0,Y 573.291,Z 324.076,A -85,B 0,C 180,E1 -2165.628,E2 -2165.628} C_VEL
LIN {X 0,Y 573.278,Z 324.073,A -85,B 0,C 180,E1 -2167.75,E2 -2167.75} C_VEL
LIN {X 0,Y 573.273,Z 324.078,A -85,B 0,C 180,E1 -2170.597,E2 -2170.597} C_VEL
LIN {X 0,Y 573.269,Z 324.078,A -85,B 0,C 180,E1 -2172.749,E2 -2172.749} C_VEL
LIN {X 0,Y 573.239,Z 324.077,A -85,B 0,C 180,E1 -2174.92,E2 -2174.92} C_VEL
LIN {X 0,Y 573.257,Z 324.082,A -85,B 0,C 180,E1 -2177.848,E2 -2177.848} C_VEL
LIN {X 0,Y 573.257,Z 324.076,A -85,B 0,C 180,E1 -2180.077,E2 -2180.077} C_VEL
LIN {X 0,Y 573.241,Z 324.083,A -85,B 0,C 180,E1 -2183.099,E2 -2183.099} C_VEL
LIN {X 0,Y 573.254,Z 324.077,A -85,B 0,C 180,E1 -2185.41,E2 -2185.41} C_VEL
LIN {X 0,Y 573.258,Z 324.076,A -85,B 0,C 180,E1 -2188.029,E2 -2188.029} C_VEL
LIN {X 0,Y 573.252,Z 324.082,A -85,B 0,C 180,E1 -2190.176,E2 -2190.176} C_VEL
LIN {X 0,Y 573.257,Z 324.074,A -85,B 0,C 180,E1 -2192.645,E2 -2192.645} C_VEL
LIN {X 0,Y 573.259,Z 324.077,A -85,B 0,C 180,E1 -2195.184,E2 -2195.184} C_VEL
LIN {X 0,Y 573.241,Z 324.078,A -85,B 0,C 180,E1 -2197.807,E2 -2197.807} C_VEL
LIN {X 0,Y 573.249,Z 324.079,A -85,B 0,C 180,E1 -2200.525,E2 -2200.525} C_VEL
LIN {X 0,Y 573.244,Z 324.076,A -85,B 0,C 180,E1 -2203.359,E2 -2203.359} C_VEL
LIN {X 0,Y 573.258,Z 324.08,A -85,B 0,C 180,E1 -2206.33,E2 -2206.33} C_VEL
LIN {X 0,Y 573.248,Z 324.077,A -85,B 0,C 180,E1 -2208.544,E2 -2208.544} C_VEL
LIN {X 0,Y 573.245,Z 324.083,A -85,B 0,C 180,E1 -2211.298,E2 -2211.298} C_VEL
LIN {X 0,Y 573.284,Z 324.173,A -85,B 0,C 180,E1 -2213.134,E2 -2213.134} C_VEL
LIN {X 0,Y 574.188,Z 329.064,A -85,B 0,C 180,E1 -2214.235,E2 -2214.235} C_VEL
LIN {X 0,Y 574.044,Z 340.132,A -85,B 0,C 180,E1 -2216.569,E2 -2216.569} C_VEL
LIN {X 0,Y 573.925,Z 353.41,A -85,B 0,C 180,E1 -2219.253,E2 -2219.253} C_VEL
LIN {X 0,Y 573.924,Z 369.023,A -85,B 0,C 180,E1 -2222.268,E2 -2222.268} C_VEL
LIN {X 0,Y 573.829,Z 383.465,A -85,B 0,C 180,E1 -2225.002,E2 -2225.002} C_VEL
LIN {X 0,Y 573.658,Z 397.188,A -85,B 0,C 180,E1 -2227.679,E2 -2227.679} C_VEL
LIN {X 0,Y 573.516,Z 410.885,A -85,B 0,C 180,E1 -2230.306,E2 -2230.306} C_VEL
LIN {X 0,Y 573.39,Z 424.88,A -85,B 0,C 180,E1 -2232.949,E2 -2232.949} C_VEL
LIN {X 0,Y 573.249,Z 440.229,A -85,B 0,C 180,E1 -2235.806,E2 -2235.806} C_VEL
LIN {X 0,Y 573.208,Z 449.11,A -85,B 0,C 180,E1 -2237.444,E2 -2237.444} C_VEL
LIN {X 0,Y 573.902,Z 454.938,A -85,B 0,C 180,E1 -2237.558,E2 -2237.558} C_VEL
LIN {X 0,Y 573.811,Z 468.214,A -85,B 0,C 180,E1 -2237.87,E2 -2237.87} C_VEL
LIN {X 0,Y 573.698,Z 480.37,A -85,B 0,C 180,E1 -2238.294,E2 -2238.294} C_VEL
LIN {X 0,Y 573.587,Z 492.632,A -85,B 0,C 180,E1 -2238.873,E2 -2238.873} C_VEL
LIN {X 0,Y 573.433,Z 504.201,A -85,B 0,C 180,E1 -2239.585,E2 -2239.585} C_VEL
LIN {X 0,Y 573.334,Z 514.598,A -85,B 0,C 180,E1 -2240.385,E2 -2240.385} C_VEL
LIN {X 0,Y 573.241,Z 523.111,A -85,B 0,C 180,E1 -2241.184,E2 -2241.184} C_VEL
LIN {X 0,Y 573.161,Z 530.96,A -85,B 0,C 180,E1 -2242.071,E2 -2242.071} C_VEL
LIN {X 0,Y 573.073,Z 538.954,A -85,B 0,C 180,E1 -2243.185,E2 -2243.185} C_VEL
LIN {X 0,Y 573.07,Z 545.68,A -85,B 0,C 180,E1 -2244.37,E2 -2244.37} C_VEL
LIN {X 0,Y 573.028,Z 550.372,A -85,B 0,C 180,E1 -2245.427,E2 -2245.427} C_VEL
LIN {X 0,Y 573.022,Z 553.957,A -85,B 0,C 180,E1 -2246.484,E2 -2246.484} C_VEL
LIN {X 0,Y 572.959,Z 555.808,A -85,B 0,C 180,E1 -2247.188,E2 -2247.188} C_VEL
LIN {X 0,Y 572.939,Z 557.199,A -85,B 0,C 180,E1 -2247.891,E2 -2247.891} C_VEL
LIN {X 0,Y 572.941,Z 558.785,A -85,B 0,C 180,E1 -2249.297,E2 -2249.297} C_VEL
LIN {X 0,Y 572.938,Z 559,A -85,B 0,C 180,E1 -2250,E2 -2250} C_VEL
LIN {X 0,Y 572.946,Z 558.186,A -85,B 0,C 180,E1 -2251.406,E2 -2251.406} C_VEL
LIN {X 0,Y 572.939,Z 557.2,A -85,B 0,C 180,E1 -2252.109,E2 -2252.109} C_VEL
LIN {X 0,Y 572.959,Z 555.81,A -85,B 0,C 180,E1 -2252.812,E2 -2252.812} C_VEL
LIN {X 0,Y 573.014,Z 552.896,A -85,B 0,C 180,E1 -2253.868,E2 -2253.868} C_VEL
LIN {X 0,Y 572.963,Z 548.949,A -85,B 0,C 180,E1 -2254.926,E2 -2254.926} C_VEL
LIN {X 0,Y 573.064,Z 542.877,A -85,B 0,C 180,E1 -2256.16,E2 -2256.16} C_VEL
LIN {X 0,Y 573.119,Z 536.237,A -85,B 0,C 180,E1 -2257.221,E2 -2257.221} C_VEL
LIN {X 0,Y 573.201,Z 527.99,A -85,B 0,C 180,E1 -2258.283,E2 -2258.283} C_VEL
LIN {X 0,Y 573.287,Z 519.538,A -85,B 0,C 180,E1 -2259.17,E2 -2259.17} C_VEL
LIN {X 0,Y 573.429,Z 509.097,A -85,B 0,C 180,E1 -2260.058,E2 -2260.058} C_VEL
LIN {X 0,Y 573.546,Z 497.434,A -85,B 0,C 180,E1 -2260.853,E2 -2260.853} C_VEL
LIN {X 0,Y 573.651,Z 486.305,A -85,B 0,C 180,E1 -2261.446,E2 -2261.446} C_VEL
LIN {X 0,Y 573.75,Z 473.171,A -85,B 0,C 180,E1 -2261.974,E2 -2261.974} C_VEL
LIN {X 0,Y 573.855,Z 460.517,A -85,B 0,C 180,E1 -2262.331,E2 -2262.331} C_VEL
LIN {X 0,Y 573.68,Z 452.106,A -85,B 0,C 180,E1 -2262.492,E2 -2262.492} C_VEL
LIN {X 0,Y 573.211,Z 449.034,A -85,B 0,C 180,E1 -2262.57,E2 -2262.57} C_VEL
LIN {X 0,Y 573.322,Z 432.404,A -85,B 0,C 180,E1 -2265.646,E2 -2265.646} C_VEL
LIN {X 0,Y 573.458,Z 418.709,A -85,B 0,C 180,E1 -2268.211,E2 -2268.211} C_VEL
LIN {X 0,Y 573.615,Z 403.54,A -85,B 0,C 180,E1 -2271.096,E2 -2271.096} C_VEL
LIN {X 0,Y 573.774,Z 389.363,A -85,B 0,C 180,E1 -2273.842,E2 -2273.842} C_VEL
LIN {X 0,Y 573.839,Z 379.202,A -85,B 0,C 180,E1 -2275.772,E2 -2275.772} C_VEL
LIN {X 0,Y 573.719,Z 363.494,A -85,B 0,C 180,E1 -2278.539,E2 -2278.539} C_VEL
LIN {X 0,Y 573.559,Z 347.7,A -85,B 0,C 180,E1 -2281.384,E2 -2281.384} C_VEL
LIN {X 0,Y 573.645,Z 329.387,A -85,B 0,C 180,E1 -2284.83,E2 -2284.83} C_VEL
LIN {X 0,Y 573.557,Z 325.69,A -85,B 0,C 180,E1 -2285.565,E2 -2285.565} C_VEL
LIN {X 0,Y 573.287,Z 324.078,A -85,B 0,C 180,E1 -2285.93,E2 -2285.93} C_VEL
LIN {X 0,Y 573.247,Z 324.083,A -85,B 0,C 180,E1 -2288.702,E2 -2288.702} C_VEL
LIN {X 0,Y 573.258,Z 324.082,A -85,B 0,C 180,E1 -2291.596,E2 -2291.596} C_VEL
LIN {X 0,Y 573.24,Z 324.083,A -85,B 0,C 180,E1 -2294.333,E2 -2294.333} C_VEL
LIN {X 0,Y 573.244,Z 324.083,A -85,B 0,C 180,E1 -2297.359,E2 -2297.359} C_VEL
LIN {X 0,Y 573.245,Z 324.08,A -85,B 0,C 180,E1 -2300.392,E2 -2300.392} C_VEL
LIN {X 0,Y 573.257,Z 324.08,A -85,B 0,C 180,E1 -2303.078,E2 -2303.078} C_VEL
LIN {X 0,Y 573.276,Z 324.079,A -85,B 0,C 180,E1 -2305.672,E2 -2305.672} C_VEL
LIN {X 0,Y 573.253,Z 324.079,A -85,B 0,C 180,E1 -2308.185,E2 -2308.185} C_VEL
LIN {X 0,Y 573.269,Z 324.075,A -85,B 0,C 180,E1 -2310.634,E2 -2310.634} C_VEL
LIN {X 0,Y 573.256,Z 324.079,A -85,B 0,C 180,E1 -2313.024,E2 -2313.024} C_VEL
LIN {X 0,Y 573.28,Z 324.077,A -85,B 0,C 180,E1 -2315.366,E2 -2315.366} C_VEL
LIN {X 0,Y 573.234,Z 324.085,A -85,B 0,C 180,E1 -2318.419,E2 -2318.419} C_VEL
LIN {X 0,Y 573.275,Z 324.076,A -85,B 0,C 180,E1 -2320.731,E2 -2320.731} C_VEL
LIN {X 0,Y 573.25,Z 324.08,A -85,B 0,C 180,E1 -2323.622,E2 -2323.622} C_VEL
LIN {X 0,Y 573.279,Z 324.076,A -85,B 0,C 180,E1 -2325.807,E2 -2325.807} C_VEL
LIN {X 0,Y 573.28,Z 324.173,A -85,B 0,C 180,E1 -2327.094,E2 -2327.094} C_VEL
LIN {X 0,Y 573.724,Z 327.294,A -85,B 0,C 180,E1 -2327.217,E2 -2327.217} C_VEL
LIN {X 0,Y 573.62,Z 338.585,A -85,B 0,C 180,E1 -2327.709,E2 -2327.709} C_VEL
LIN {X 0,Y 573.503,Z 349.72,A -85,B 0,C 180,E1 -2328.335,E2 -2328.335} C_VEL
LIN {X 0,Y 573.424,Z 360.464,A -85,B 0,C 180,E1 -2329.092,E2 -2329.092} C_VEL
LIN {X 0,Y 573.273,Z 370.196,A -85,B 0,C 180,E1 -2329.939,E2 -2329.939} C_VEL
LIN {X 0,Y 573.202,Z 378.55,A -85,B 0,C 180,E1 -2330.828,E2 -2330.828} C_VEL
LIN {X 0,Y 573.127,Z 386.727,A -85,B 0,C 180,E1 -2331.893,E2 -2331.893} C_VEL
LIN {X 0,Y 573.058,Z 393.286,A -85,B 0,C 180,E1 -2332.955,E2 -2332.955} C_VEL
LIN {X 0,Y 573.032,Z 398.496,A -85,B 0,C 180,E1 -2334.016,E2 -2334.016} C_VEL
LIN {X 0,Y 572.953,Z 402.549,A -85,B 0,C 180,E1 -2335.074,E2 -2335.074} C_VEL
LIN {X 0,Y 573.031,Z 404.679,A -85,B 0,C 180,E1 -2335.78,E2 -2335.78} C_VEL
LIN {X 0,Y 573.01,Z 406.342,A -85,B 0,C 180,E1 -2336.484,E2 -2336.484} C_VEL
LIN {X 0,Y 572.936,Z 408.461,A -85,B 0,C 180,E1 -2337.891,E2 -2337.891} C_VEL
LIN {X 0,Y 572.947,Z 408.908,A -85,B 0,C 180,E1 -2338.594,E2 -2338.594} C_VEL
LIN {X 0,Y 572.939,Z 408.618,A -85,B 0,C 180,E1 -2340,E2 -2340} C_VEL
LIN {X 0,Y 572.942,Z 407.897,A -85,B 0,C 180,E1 -2340.703,E2 -2340.703} C_VEL
LIN {X 0,Y 572.949,Z 406.742,A -85,B 0,C 180,E1 -2341.406,E2 -2341.406} C_VEL
LIN {X 0,Y 572.947,Z 405.187,A -85,B 0,C 180,E1 -2342.109,E2 -2342.109} C_VEL
LIN {X 0,Y 573.011,Z 402.045,A -85,B 0,C 180,E1 -2343.164,E2 -2343.164} C_VEL
LIN {X 0,Y 573.036,Z 397.85,A -85,B 0,C 180,E1 -2344.22,E2 -2344.22} C_VEL
LIN {X 0,Y 573.054,Z 391.459,A -85,B 0,C 180,E1 -2345.454,E2 -2345.454} C_VEL
LIN {X 0,Y 573.155,Z 383.886,A -85,B 0,C 180,E1 -2346.595,E2 -2346.595} C_VEL
LIN {X 0,Y 573.22,Z 375.798,A -85,B 0,C 180,E1 -2347.574,E2 -2347.574} C_VEL
LIN {X 0,Y 573.337,Z 365.902,A -85,B 0,C 180,E1 -2348.547,E2 -2348.547} C_VEL
LIN {X 0,Y 573.427,Z 355.833,A -85,B 0,C 180,E1 -2349.346,E2 -2349.346} C_VEL
LIN {X 0,Y 573.569,Z 344.695,A -85,B 0,C 180,E1 -2350.056,E2 -2350.056} C_VEL
LIN {X 0,Y 573.667,Z 332.547,A -85,B 0,C 180,E1 -2350.662,E2 -2350.662} C_VEL
LIN {X 0,Y 573.594,Z 325.7,A -85,B 0,C 180,E1 -2350.935,E2 -2350.935} C_VEL
LIN {X 0,Y 573.258,Z 324.076,A -85,B 0,C 180,E1 -2351.022,E2 -2351.022} C_VEL
LIN {X 0,Y 573.24,Z 324.081,A -85,B 0,C 180,E1 -2353.47,E2 -2353.47} C_VEL
LIN {X 0,Y 573.241,Z 324.083,A -85,B 0,C 180,E1 -2355.648,E2 -2355.648} C_VEL
LIN {X 0,Y 573.244,Z 324.077,A -85,B 0,C 180,E1 -2357.848,E2 -2357.848} C_VEL
LIN {X 0,Y 573.247,Z 324.075,A -85,B 0,C 180,E1 -2360.077,E2 -2360.077} C_VEL
LIN {X 0,Y 573.224,Z 324.079,A -85,B 0,C 180,E1 -2361.9,E2 -2361.9} C_VEL
LIN {X 0,Y 572.592,Z 324.163,A -85,B 0,C 180,E1 -2362.486,E2 -2362.486} C_VEL
LIN {X 0,Y 569.839,Z 324.505,A -85,B 0,C 180,E1 -2363.438,E2 -2363.438} C_VEL
LIN {X 0,Y 567.455,Z 324.802,A -85,B 0,C 180,E1 -2364.203,E2 -2364.203} C_VEL
LIN {X 0,Y 566.36,Z 324.937,A -85,B 0,C 180,E1 -2364.794,E2 -2364.794} C_VEL
LIN {X 0,Y 566.232,Z 324.951,A -85,B 0,C 180,E1 -2364.993,E2 -2364.993} C_VEL
